// TIA Portal V20 export
// export: Created 2025-12-01T14:57:42.4272201Z, ExportSetting None, DisplayName Totally Integrated Automation Portal, DisplayVersion V20 Update 3, DisplayName TIA Portal Openness, DisplayVersion V20 Update 3, DisplayName TIA Portal Version Control Interface, DisplayVersion V20 Update 3, DisplayName STEP 7 Professional, DisplayVersion V20 Update 3, DisplayName STEP 7 Safety, DisplayVersion V20 Update 2, DisplayName WinCC Basic/Comfort/Advanced, DisplayVersion V20 Update 3, DisplayName WinCC Professional, DisplayVersion V20 Update 3, DisplayName WinCC Unified, DisplayVersion V20 Update 3
DATA_BLOCK "DB5_Emison"   // DB5
{ S7_Optimized_Access := 'FALSE' }
// stored: AutoNumber false
   VAR
      ByteLIbre_000 : Byte;
      RecepOK_M1 : Bool;
      PresNormal_M1 : Bool;
      Ausencia_M1 : Bool;
      PresBloqueo_M1 : Bool;
      Galibo_M1 : Bool;
      PresPreparada_M1 : Bool;
      PresMultiple_M1 : Bool;
      Bit_07_M1 : Bool;
      RecepOK_M2 : Bool;
      PresNormal_M2 : Bool;
      Ausencia_M2 : Bool;
      PresBloqueo_M2 : Bool;
      Galibo_M2 : Bool;
      PresPreparada_M2 : Bool;
      PresMultiple_M2 : Bool;
      Bit_07_M2 : Bool;
      RecepOK_M3 : Bool;
      PresNormal_M3 : Bool;
      Ausencia_M3 : Bool;
      PresBloqueo_M3 : Bool;
      Galibo_M3 : Bool;
      PresPreparada_M3 : Bool;
      PresMultiple_M3 : Bool;
      Bit_07_M3 : Bool;
      RecepOK_M4 : Bool;
      PresNormal_M4 : Bool;
      Ausencia_M4 : Bool;
      PresBloqueo_M4 : Bool;
      Galibo_M4 : Bool;
      PresPreparada_M4 : Bool;
      PresMultiple_M4 : Bool;
      Bit_07_M4 : Bool;
      RecepOK_M5 : Bool;
      PresNormal_M5 : Bool;
      Ausencia_M5 : Bool;
      PresBloqueo_M5 : Bool;
      Galibo_M5 : Bool;
      PresPreparada_M5 : Bool;
      PresMultiple_M5 : Bool;
      Bit_07_M5 : Bool;
      RecepOK_M6 : Bool;
      PresNormal_M6 : Bool;
      Ausencia_M6 : Bool;
      PresBloqueo_M6 : Bool;
      Galibo_M6 : Bool;
      PresPreparada_M6 : Bool;
      PresMultiple_M6 : Bool;
      Bit_07_M6 : Bool;
      RecepOK_M7 : Bool;
      PresNormal_M7 : Bool;
      Ausencia_M7 : Bool;
      PresBloqueo_M7 : Bool;
      Galibo_M7 : Bool;
      PresPreparada_M7 : Bool;
      PresMultiple_M7 : Bool;
      Bit_07_M7 : Bool;
      RecepOK_M8 : Bool;
      PresNormal_M8 : Bool;
      Ausencia_M8 : Bool;
      PresBloqueo_M8 : Bool;
      Galibo_M8 : Bool;
      PresPreparada_M8 : Bool;
      PresMultiple_M8 : Bool;
      Bit_07_M8 : Bool;
      RecepOK_M9 : Bool;
      PresNormal_M9 : Bool;
      Ausencia_M9 : Bool;
      PresBloqueo_M9 : Bool;
      Galibo_M9 : Bool;
      PresPreparada_M9 : Bool;
      PresMultiple_M9 : Bool;
      Bit_07_M9 : Bool;
      RecepOK_M10 : Bool;
      PresNormal_M10 : Bool;
      Ausencia_M10 : Bool;
      PresBloqueo_M10 : Bool;
      Galibo_M10 : Bool;
      PresPreparada_M10 : Bool;
      PresMultiple_M10 : Bool;
      Bit_07_M10 : Bool;
      RecepOK_M11 : Bool;
      PresNormal_M11 : Bool;
      Ausencia_M11 : Bool;
      PresBloqueo_M11 : Bool;
      Galibo_M11 : Bool;
      PresPreparada_M11 : Bool;
      PresMultiple_M11 : Bool;
      Bit_07_M11 : Bool;
      RecepOK_M12 : Bool;
      PresNormal_M12 : Bool;
      Ausencia_M12 : Bool;
      PresBloqueo_M12 : Bool;
      Galibo_M12 : Bool;
      PresPreparada_M12 : Bool;
      PresMultiple_M12 : Bool;
      Bit_07_M12 : Bool;
      RecepOK_M13 : Bool;
      PresNormal_M13 : Bool;
      Ausencia_M13 : Bool;
      PresBloqueo_M13 : Bool;
      Galibo_M13 : Bool;
      PresPreparada_M13 : Bool;
      PresMultiple_M13 : Bool;
      Bit_07_M13 : Bool;
      RecepOK_M14 : Bool;
      PresNormal_M14 : Bool;
      Ausencia_M14 : Bool;
      PresBloqueo_M14 : Bool;
      Galibo_M14 : Bool;
      PresPreparada_M14 : Bool;
      PresMultiple_M14 : Bool;
      Bit_07_M14 : Bool;
      RecepOK_M15 : Bool;
      PresNormal_M15 : Bool;
      Ausencia_M15 : Bool;
      PresBloqueo_M15 : Bool;
      Galibo_M15 : Bool;
      PresPreparada_M15 : Bool;
      PresMultiple_M15 : Bool;
      Bit_07_M15 : Bool;
      RecepOK_M16 : Bool;
      PresNormal_M16 : Bool;
      Ausencia_M16 : Bool;
      PresBloqueo_M16 : Bool;
      Galibo_M16 : Bool;
      PresPreparada_M16 : Bool;
      PresMultiple_M16 : Bool;
      Bit_07_M16 : Bool;
      RecepOK_M17 : Bool;
      PresNormal_M17 : Bool;
      Ausencia_M17 : Bool;
      PresBloqueo_M17 : Bool;
      Galibo_M17 : Bool;
      PresPreparada_M17 : Bool;
      PresMultiple_M17 : Bool;
      Bit_07_M17 : Bool;
      RecepOK_M18 : Bool;
      PresNormal_M18 : Bool;
      Ausencia_M18 : Bool;
      PresBloqueo_M18 : Bool;
      Galibo_M18 : Bool;
      PresPreparada_M18 : Bool;
      PresMultiple_M18 : Bool;
      Bit_07_M18 : Bool;
      RecepOK_M19 : Bool;
      PresNormal_M19 : Bool;
      Ausencia_M19 : Bool;
      PresBloqueo_M19 : Bool;
      Galibo_M19 : Bool;
      PresPreparada_M19 : Bool;
      PresMultiple_M19 : Bool;
      Bit_07_M19 : Bool;
      RecepOK_M20 : Bool;
      PresNormal_M20 : Bool;
      Ausencia_M20 : Bool;
      PresBloqueo_M20 : Bool;
      Galibo_M20 : Bool;
      PresPreparada_M20 : Bool;
      PresMultiple_M20 : Bool;
      Bit_07_M20 : Bool;
      RecepOK_M21 : Bool;
      PresNormal_M21 : Bool;
      Ausencia_M21 : Bool;
      PresBloqueo_M21 : Bool;
      Galibo_M21 : Bool;
      PresPreparada_M21 : Bool;
      PresMultiple_M21 : Bool;
      Bit_07_M21 : Bool;
      RecepOK_M22 : Bool;
      PresNormal_M22 : Bool;
      Ausencia_M22 : Bool;
      PresBloqueo_M22 : Bool;
      Galibo_M22 : Bool;
      PresPreparada_M22 : Bool;
      PresMultiple_M22 : Bool;
      Bit_07_M22 : Bool;
      RecepOK_M23 : Bool;
      PresNormal_M23 : Bool;
      Ausencia_M23 : Bool;
      PresBloqueo_M23 : Bool;
      Galibo_M23 : Bool;
      PresPreparada_M23 : Bool;
      PresMultiple_M23 : Bool;
      Bit_07_M23 : Bool;
      RecepOK_M24 : Bool;
      PresNormal_M24 : Bool;
      Ausencia_M24 : Bool;
      PresBloqueo_M24 : Bool;
      Galibo_M24 : Bool;
      PresPreparada_M24 : Bool;
      PresMultiple_M24 : Bool;
      Bit_07_M24 : Bool;
      RecepOK_M25 : Bool;
      PresNormal_M25 : Bool;
      Ausencia_M25 : Bool;
      PresBloqueo_M25 : Bool;
      Galibo_M25 : Bool;
      PresPreparada_M25 : Bool;
      PresMultiple_M25 : Bool;
      Bit_07_M25 : Bool;
      RecepOK_M26 : Bool;
      PresNormal_M26 : Bool;
      Ausencia_M26 : Bool;
      PresBloqueo_M26 : Bool;
      Galibo_M26 : Bool;
      PresPreparada_M26 : Bool;
      PresMultiple_M26 : Bool;
      Bit_07_M26 : Bool;
      RecepOK_M27 : Bool;
      PresNormal_M27 : Bool;
      Ausencia_M27 : Bool;
      PresBloqueo_M27 : Bool;
      Galibo_M27 : Bool;
      PresPreparada_M27 : Bool;
      PresMultiple_M27 : Bool;
      Bit_07_M27 : Bool;
      RecepOK_M28 : Bool;
      PresNormal_M28 : Bool;
      Ausencia_M28 : Bool;
      PresBloqueo_M28 : Bool;
      Galibo_M28 : Bool;
      PresPreparada_M28 : Bool;
      PresMultiple_M28 : Bool;
      Bit_07_M28 : Bool;
      RecepOK_M29 : Bool;
      PresNormal_M29 : Bool;
      Ausencia_M29 : Bool;
      PresBloqueo_M29 : Bool;
      Galibo_M29 : Bool;
      PresPreparada_M29 : Bool;
      PresMultiple_M29 : Bool;
      Bit_07_M29 : Bool;
      RecepOK_M30 : Bool;
      PresNormal_M30 : Bool;
      Ausencia_M30 : Bool;
      PresBloqueo_M30 : Bool;
      Galibo_M30 : Bool;
      PresPreparada_M30 : Bool;
      PresMultiple_M30 : Bool;
      Bit_07_M30 : Bool;
      RecepOK_M31 : Bool;
      PresNormal_M31 : Bool;
      Ausencia_M31 : Bool;
      PresBloqueo_M31 : Bool;
      Galibo_M31 : Bool;
      PresPreparada_M31 : Bool;
      PresMultiple_M31 : Bool;
      Bit_07_M31 : Bool;
      RecepOK_M32 : Bool;
      PresNormal_M32 : Bool;
      Ausencia_M32 : Bool;
      PresBloqueo_M32 : Bool;
      Galibo_M32 : Bool;
      PresPreparada_M32 : Bool;
      PresMultiple_M32 : Bool;
      Bit_07_M32 : Bool;
      RecepOK_M33 : Bool;
      PresNormal_M33 : Bool;
      Ausencia_M33 : Bool;
      PresBloqueo_M33 : Bool;
      Galibo_M33 : Bool;
      PresPreparada_M33 : Bool;
      PresMultiple_M33 : Bool;
      Bit_07_M33 : Bool;
      RecepOK_M34 : Bool;
      PresNormal_M34 : Bool;
      Ausencia_M34 : Bool;
      PresBloqueo_M34 : Bool;
      Galibo_M34 : Bool;
      PresPreparada_M34 : Bool;
      PresMultiple_M34 : Bool;
      Bit_07_M34 : Bool;
      RecepOK_M35 : Bool;
      PresNormal_M35 : Bool;
      Ausencia_M35 : Bool;
      PresBloqueo_M35 : Bool;
      Galibo_M35 : Bool;
      PresPreparada_M35 : Bool;
      PresMultiple_M35 : Bool;
      Bit_07_M35 : Bool;
      RecepOK_M36 : Bool;
      PresNormal_M36 : Bool;
      Ausencia_M36 : Bool;
      PresBloqueo_M36 : Bool;
      Galibo_M36 : Bool;
      PresPreparada_M36 : Bool;
      PresMultiple_M36 : Bool;
      Bit_07_M36 : Bool;
      RecepOK_M37 : Bool;
      PresNormal_M37 : Bool;
      Ausencia_M37 : Bool;
      PresBloqueo_M37 : Bool;
      Galibo_M37 : Bool;
      PresPreparada_M37 : Bool;
      PresMultiple_M37 : Bool;
      Bit_07_M37 : Bool;
      RecepOK_M38 : Bool;
      PresNormal_M38 : Bool;
      Ausencia_M38 : Bool;
      PresBloqueo_M38 : Bool;
      Galibo_M38 : Bool;
      PresPreparada_M38 : Bool;
      PresMultiple_M38 : Bool;
      Bit_07_M38 : Bool;
      RecepOK_M39 : Bool;
      PresNormal_M39 : Bool;
      Ausencia_M39 : Bool;
      PresBloqueo_M39 : Bool;
      Galibo_M39 : Bool;
      PresPreparada_M39 : Bool;
      PresMultiple_M39 : Bool;
      Bit_07_M39 : Bool;
      RecepOK_M40 : Bool;
      PresNormal_M40 : Bool;
      Ausencia_M40 : Bool;
      PresBloqueo_M40 : Bool;
      Galibo_M40 : Bool;
      PresPreparada_M40 : Bool;
      PresMultiple_M40 : Bool;
      Bit_07_M40 : Bool;
      RecepOK_M41 : Bool;
      PresNormal_M41 : Bool;
      Ausencia_M41 : Bool;
      PresBloqueo_M41 : Bool;
      Galibo_M41 : Bool;
      PresPreparada_M41 : Bool;
      PresMultiple_M41 : Bool;
      Bit_07_M41 : Bool;
      RecepOK_M42 : Bool;
      PresNormal_M42 : Bool;
      Ausencia_M42 : Bool;
      PresBloqueo_M42 : Bool;
      Galibo_M42 : Bool;
      PresPreparada_M42 : Bool;
      PresMultiple_M42 : Bool;
      Bit_07_M42 : Bool;
      RecepOK_M43 : Bool;
      PresNormal_M43 : Bool;
      Ausencia_M43 : Bool;
      PresBloqueo_M43 : Bool;
      Galibo_M43 : Bool;
      PresPreparada_M43 : Bool;
      PresMultiple_M43 : Bool;
      Bit_07_M43 : Bool;
      RecepOK_M44 : Bool;
      PresNormal_M44 : Bool;
      Ausencia_M44 : Bool;
      PresBloqueo_M44 : Bool;
      Galibo_M44 : Bool;
      PresPreparada_M44 : Bool;
      PresMultiple_M44 : Bool;
      Bit_07_M44 : Bool;
      RecepOK_M45 : Bool;
      PresNormal_M45 : Bool;
      Ausencia_M45 : Bool;
      PresBloqueo_M45 : Bool;
      Galibo_M45 : Bool;
      PresPreparada_M45 : Bool;
      PresMultiple_M45 : Bool;
      Bit_07_M45 : Bool;
      RecepOK_M46 : Bool;
      PresNormal_M46 : Bool;
      Ausencia_M46 : Bool;
      PresBloqueo_M46 : Bool;
      Galibo_M46 : Bool;
      PresPreparada_M46 : Bool;
      PresMultiple_M46 : Bool;
      Bit_07_M46 : Bool;
      RecepOK_M47 : Bool;
      PresNormal_M47 : Bool;
      Ausencia_M47 : Bool;
      PresBloqueo_M47 : Bool;
      Galibo_M47 : Bool;
      PresPreparada_M47 : Bool;
      PresMultiple_M47 : Bool;
      Bit_07_M47 : Bool;
      RecepOK_M48 : Bool;
      PresNormal_M48 : Bool;
      Ausencia_M48 : Bool;
      PresBloqueo_M48 : Bool;
      Galibo_M48 : Bool;
      PresPreparada_M48 : Bool;
      PresMultiple_M48 : Bool;
      Bit_07_M48 : Bool;
      RecepOK_M49 : Bool;
      PresNormal_M49 : Bool;
      Ausencia_M49 : Bool;
      PresBloqueo_M49 : Bool;
      Galibo_M49 : Bool;
      PresPreparada_M49 : Bool;
      PresMultiple_M49 : Bool;
      Bit_07_M49 : Bool;
      RecepOK_M50 : Bool;
      PresNormal_M50 : Bool;
      Ausencia_M50 : Bool;
      PresBloqueo_M50 : Bool;
      Galibo_M50 : Bool;
      PresPreparada_M50 : Bool;
      PresMultiple_M50 : Bool;
      Bit_07_M50 : Bool;
      RecepOK_M51 : Bool;
      PresNormal_M51 : Bool;
      Ausencia_M51 : Bool;
      PresBloqueo_M51 : Bool;
      Galibo_M51 : Bool;
      PresPreparada_M51 : Bool;
      PresMultiple_M51 : Bool;
      Bit_07_M51 : Bool;
      RecepOK_M52 : Bool;
      PresNormal_M52 : Bool;
      Ausencia_M52 : Bool;
      PresBloqueo_M52 : Bool;
      Galibo_M52 : Bool;
      PresPreparada_M52 : Bool;
      PresMultiple_M52 : Bool;
      Bit_07_M52 : Bool;
      RecepOK_M53 : Bool;
      PresNormal_M53 : Bool;
      Ausencia_M53 : Bool;
      PresBloqueo_M53 : Bool;
      Galibo_M53 : Bool;
      PresPreparada_M53 : Bool;
      PresMultiple_M53 : Bool;
      Bit_07_M53 : Bool;
      RecepOK_M54 : Bool;
      PresNormal_M54 : Bool;
      Ausencia_M54 : Bool;
      PresBloqueo_M54 : Bool;
      Galibo_M54 : Bool;
      PresPreparada_M54 : Bool;
      PresMultiple_M54 : Bool;
      Bit_07_M54 : Bool;
      RecepOK_M55 : Bool;
      PresNormal_M55 : Bool;
      Ausencia_M55 : Bool;
      PresBloqueo_M55 : Bool;
      Galibo_M55 : Bool;
      PresPreparada_M55 : Bool;
      PresMultiple_M55 : Bool;
      Bit_07_M55 : Bool;
      RecepOK_M56 : Bool;
      PresNormal_M56 : Bool;
      Ausencia_M56 : Bool;
      PresBloqueo_M56 : Bool;
      Galibo_M56 : Bool;
      PresPreparada_M56 : Bool;
      PresMultiple_M56 : Bool;
      Bit_07_M56 : Bool;
      RecepOK_M57 : Bool;
      PresNormal_M57 : Bool;
      Ausencia_M57 : Bool;
      PresBloqueo_M57 : Bool;
      Galibo_M57 : Bool;
      PresPreparada_M57 : Bool;
      PresMultiple_M57 : Bool;
      Bit_07_M57 : Bool;
      RecepOK_M58 : Bool;
      PresNormal_M58 : Bool;
      Ausencia_M58 : Bool;
      PresBloqueo_M58 : Bool;
      Galibo_M58 : Bool;
      PresPreparada_M58 : Bool;
      PresMultiple_M58 : Bool;
      Bit_07_M58 : Bool;
      RecepOK_M59 : Bool;
      PresNormal_M59 : Bool;
      Ausencia_M59 : Bool;
      PresBloqueo_M59 : Bool;
      Galibo_M59 : Bool;
      PresPreparada_M59 : Bool;
      PresMultiple_M59 : Bool;
      Bit_07_M59 : Bool;
      RecepOK_M60 : Bool;
      PresNormal_M60 : Bool;
      Ausencia_M60 : Bool;
      PresBloqueo_M60 : Bool;
      Galibo_M60 : Bool;
      PresPreparada_M60 : Bool;
      PresMultiple_M60 : Bool;
      Bit_07_M60 : Bool;
      RecepOK_M61 : Bool;
      PresNormal_M61 : Bool;
      Ausencia_M61 : Bool;
      PresBloqueo_M61 : Bool;
      Galibo_M61 : Bool;
      PresPreparada_M61 : Bool;
      PresMultiple_M61 : Bool;
      Bit_07_M61 : Bool;
      RecepOK_M62 : Bool;
      PresNormal_M62 : Bool;
      Ausencia_M62 : Bool;
      PresBloqueo_M62 : Bool;
      Galibo_M62 : Bool;
      PresPreparada_M62 : Bool;
      PresMultiple_M62 : Bool;
      Bit_07_M62 : Bool;
      RecepOK_M63 : Bool;
      PresNormal_M63 : Bool;
      Ausencia_M63 : Bool;
      PresBloqueo_M63 : Bool;
      Galibo_M63 : Bool;
      PresPreparada_M63 : Bool;
      PresMultiple_M63 : Bool;
      Bit_07_M63 : Bool;
      RecepOK_M64 : Bool;
      PresNormal_M64 : Bool;
      Ausencia_M64 : Bool;
      PresBloqueo_M64 : Bool;
      Galibo_M64 : Bool;
      PresPreparada_M64 : Bool;
      PresMultiple_M64 : Bool;
      Bit_07_M64 : Bool;
      RecepOK_M65 : Bool;
      PresNormal_M65 : Bool;
      Ausencia_M65 : Bool;
      PresBloqueo_M65 : Bool;
      Galibo_M65 : Bool;
      PresPreparada_M65 : Bool;
      PresMultiple_M65 : Bool;
      Bit_07_M65 : Bool;
      RecepOK_M66 : Bool;
      PresNormal_M66 : Bool;
      Ausencia_M66 : Bool;
      PresBloqueo_M66 : Bool;
      Galibo_M66 : Bool;
      PresPreparada_M66 : Bool;
      PresMultiple_M66 : Bool;
      Bit_07_M66 : Bool;
      RecepOK_M67 : Bool;
      PresNormal_M67 : Bool;
      Ausencia_M67 : Bool;
      PresBloqueo_M67 : Bool;
      Galibo_M67 : Bool;
      PresPreparada_M67 : Bool;
      PresMultiple_M67 : Bool;
      Bit_07_M67 : Bool;
      RecepOK_M68 : Bool;
      PresNormal_M68 : Bool;
      Ausencia_M68 : Bool;
      PresBloqueo_M68 : Bool;
      Galibo_M68 : Bool;
      PresPreparada_M68 : Bool;
      PresMultiple_M68 : Bool;
      Bit_07_M68 : Bool;
      RecepOK_M69 : Bool;
      PresNormal_M69 : Bool;
      Ausencia_M69 : Bool;
      PresBloqueo_M69 : Bool;
      Galibo_M69 : Bool;
      PresPreparada_M69 : Bool;
      PresMultiple_M69 : Bool;
      Bit_07_M69 : Bool;
      RecepOK_M70 : Bool;
      PresNormal_M70 : Bool;
      Ausencia_M70 : Bool;
      PresBloqueo_M70 : Bool;
      Galibo_M70 : Bool;
      PresPreparada_M70 : Bool;
      PresMultiple_M70 : Bool;
      Bit_07_M70 : Bool;
      RecepOK_M71 : Bool;
      PresNormal_M71 : Bool;
      Ausencia_M71 : Bool;
      PresBloqueo_M71 : Bool;
      Galibo_M71 : Bool;
      PresPreparada_M71 : Bool;
      PresMultiple_M71 : Bool;
      Bit_07_M71 : Bool;
      RecepOK_M72 : Bool;
      PresNormal_M72 : Bool;
      Ausencia_M72 : Bool;
      PresBloqueo_M72 : Bool;
      Galibo_M72 : Bool;
      PresPreparada_M72 : Bool;
      PresMultiple_M72 : Bool;
      Bit_07_M72 : Bool;
      RecepOK_M73 : Bool;
      PresNormal_M73 : Bool;
      Ausencia_M73 : Bool;
      PresBloqueo_M73 : Bool;
      Galibo_M73 : Bool;
      PresPreparada_M73 : Bool;
      PresMultiple_M73 : Bool;
      Bit_07_M73 : Bool;
      RecepOK_M74 : Bool;
      PresNormal_M74 : Bool;
      Ausencia_M74 : Bool;
      PresBloqueo_M74 : Bool;
      Galibo_M74 : Bool;
      PresPreparada_M74 : Bool;
      PresMultiple_M74 : Bool;
      Bit_07_M74 : Bool;
      RecepOK_M75 : Bool;
      PresNormal_M75 : Bool;
      Ausencia_M75 : Bool;
      PresBloqueo_M75 : Bool;
      Galibo_M75 : Bool;
      PresPreparada_M75 : Bool;
      PresMultiple_M75 : Bool;
      Bit_07_M75 : Bool;
      RecepOK_M76 : Bool;
      PresNormal_M76 : Bool;
      Ausencia_M76 : Bool;
      PresBloqueo_M76 : Bool;
      Galibo_M76 : Bool;
      PresPreparada_M76 : Bool;
      PresMultiple_M76 : Bool;
      Bit_07_M76 : Bool;
      RecepOK_M77 : Bool;
      PresNormal_M77 : Bool;
      Ausencia_M77 : Bool;
      PresBloqueo_M77 : Bool;
      Galibo_M77 : Bool;
      PresPreparada_M77 : Bool;
      PresMultiple_M77 : Bool;
      Bit_07_M77 : Bool;
      RecepOK_M78 : Bool;
      PresNormal_M78 : Bool;
      Ausencia_M78 : Bool;
      PresBloqueo_M78 : Bool;
      Galibo_M78 : Bool;
      PresPreparada_M78 : Bool;
      PresMultiple_M78 : Bool;
      Bit_07_M78 : Bool;
      RecepOK_M79 : Bool;
      PresNormal_M79 : Bool;
      Ausencia_M79 : Bool;
      PresBloqueo_M79 : Bool;
      Galibo_M79 : Bool;
      PresPreparada_M79 : Bool;
      PresMultiple_M79 : Bool;
      Bit_07_M79 : Bool;
      RecepOK_M80 : Bool;
      PresNormal_M80 : Bool;
      Ausencia_M80 : Bool;
      PresBloqueo_M80 : Bool;
      Galibo_M80 : Bool;
      PresPreparada_M80 : Bool;
      PresMultiple_M80 : Bool;
      Bit_07_M80 : Bool;
      RecepOK_M81 : Bool;
      PresNormal_M81 : Bool;
      Ausencia_M81 : Bool;
      PresBloqueo_M81 : Bool;
      Galibo_M81 : Bool;
      PresPreparada_M81 : Bool;
      PresMultiple_M81 : Bool;
      Bit_07_M81 : Bool;
      RecepOK_M82 : Bool;
      PresNormal_M82 : Bool;
      Ausencia_M82 : Bool;
      PresBloqueo_M82 : Bool;
      Galibo_M82 : Bool;
      PresPreparada_M82 : Bool;
      PresMultiple_M82 : Bool;
      Bit_07_M82 : Bool;
      RecepOK_M83 : Bool;
      PresNormal_M83 : Bool;
      Ausencia_M83 : Bool;
      PresBloqueo_M83 : Bool;
      Galibo_M83 : Bool;
      PresPreparada_M83 : Bool;
      PresMultiple_M83 : Bool;
      Bit_07_M83 : Bool;
      RecepOK_M84 : Bool;
      PresNormal_M84 : Bool;
      Ausencia_M84 : Bool;
      PresBloqueo_M84 : Bool;
      Galibo_M84 : Bool;
      PresPreparada_M84 : Bool;
      PresMultiple_M84 : Bool;
      Bit_07_M84 : Bool;
      RecepOK_M85 : Bool;
      PresNormal_M85 : Bool;
      Ausencia_M85 : Bool;
      PresBloqueo_M85 : Bool;
      Galibo_M85 : Bool;
      PresPreparada_M85 : Bool;
      PresMultiple_M85 : Bool;
      Bit_07_M85 : Bool;
      RecepOK_M86 : Bool;
      PresNormal_M86 : Bool;
      Ausencia_M86 : Bool;
      PresBloqueo_M86 : Bool;
      Galibo_M86 : Bool;
      PresPreparada_M86 : Bool;
      PresMultiple_M86 : Bool;
      Bit_07_M86 : Bool;
      RecepOK_M87 : Bool;
      PresNormal_M87 : Bool;
      Ausencia_M87 : Bool;
      PresBloqueo_M87 : Bool;
      Galibo_M87 : Bool;
      PresPreparada_M87 : Bool;
      PresMultiple_M87 : Bool;
      Bit_07_M87 : Bool;
      RecepOK_M88 : Bool;
      PresNormal_M88 : Bool;
      Ausencia_M88 : Bool;
      PresBloqueo_M88 : Bool;
      Galibo_M88 : Bool;
      PresPreparada_M88 : Bool;
      PresMultiple_M88 : Bool;
      Bit_07_M88 : Bool;
      RecepOK_M89 : Bool;
      PresNormal_M89 : Bool;
      Ausencia_M89 : Bool;
      PresBloqueo_M89 : Bool;
      Galibo_M89 : Bool;
      PresPreparada_M89 : Bool;
      PresMultiple_M89 : Bool;
      Bit_07_M89 : Bool;
      RecepOK_M90 : Bool;
      PresNormal_M90 : Bool;
      Ausencia_M90 : Bool;
      PresBloqueo_M90 : Bool;
      Galibo_M90 : Bool;
      PresPreparada_M90 : Bool;
      PresMultiple_M90 : Bool;
      Bit_07_M90 : Bool;
      RecepOK_M91 : Bool;
      PresNormal_M91 : Bool;
      Ausencia_M91 : Bool;
      PresBloqueo_M91 : Bool;
      Galibo_M91 : Bool;
      PresPreparada_M91 : Bool;
      PresMultiple_M91 : Bool;
      Bit_07_M91 : Bool;
      RecepOK_M92 : Bool;
      PresNormal_M92 : Bool;
      Ausencia_M92 : Bool;
      PresBloqueo_M92 : Bool;
      Galibo_M92 : Bool;
      PresPreparada_M92 : Bool;
      PresMultiple_M92 : Bool;
      Bit_07_M92 : Bool;
      RecepOK_M93 : Bool;
      PresNormal_M93 : Bool;
      Ausencia_M93 : Bool;
      PresBloqueo_M93 : Bool;
      Galibo_M93 : Bool;
      PresPreparada_M93 : Bool;
      PresMultiple_M93 : Bool;
      Bit_07_M93 : Bool;
      RecepOK_M94 : Bool;
      PresNormal_M94 : Bool;
      Ausencia_M94 : Bool;
      PresBloqueo_M94 : Bool;
      Galibo_M94 : Bool;
      PresPreparada_M94 : Bool;
      PresMultiple_M94 : Bool;
      Bit_07_M94 : Bool;
      RecepOK_M95 : Bool;
      PresNormal_M95 : Bool;
      Ausencia_M95 : Bool;
      PresBloqueo_M95 : Bool;
      Galibo_M95 : Bool;
      PresPreparada_M95 : Bool;
      PresMultiple_M95 : Bool;
      Bit_07_M95 : Bool;
      RecepOK_M96 : Bool;
      PresNormal_M96 : Bool;
      Ausencia_M96 : Bool;
      PresBloqueo_M96 : Bool;
      Galibo_M96 : Bool;
      PresPreparada_M96 : Bool;
      PresMultiple_M96 : Bool;
      Bit_07_M96 : Bool;
      RecepOK_M97 : Bool;
      PresNormal_M97 : Bool;
      Ausencia_M97 : Bool;
      PresBloqueo_M97 : Bool;
      Galibo_M97 : Bool;
      PresPreparada_M97 : Bool;
      PresMultiple_M97 : Bool;
      Bit_07_M97 : Bool;
      RecepOK_M98 : Bool;
      PresNormal_M98 : Bool;
      Ausencia_M98 : Bool;
      PresBloqueo_M98 : Bool;
      Galibo_M98 : Bool;
      PresPreparada_M98 : Bool;
      PresMultiple_M98 : Bool;
      Bit_07_M98 : Bool;
      RecepOK_M99 : Bool;
      PresNormal_M99 : Bool;
      Ausencia_M99 : Bool;
      PresBloqueo_M99 : Bool;
      Galibo_M99 : Bool;
      PresPreparada_M99 : Bool;
      PresMultiple_M99 : Bool;
      Bit_07_M99 : Bool;
      RecepOK_M100 : Bool;
      PresNormal_M100 : Bool;
      Ausencia_M100 : Bool;
      PresBloqueo_M100 : Bool;
      Galibo_M100 : Bool;
      PresPreparada_M100 : Bool;
      PresMultiple_M100 : Bool;
      Bit_07_M100 : Bool;
      RecepOK_M101 : Bool;
      PresNormal_M101 : Bool;
      Ausencia_M101 : Bool;
      PresBloqueo_M101 : Bool;
      Galibo_M101 : Bool;
      PresPreparada_M101 : Bool;
      PresMultiple_M101 : Bool;
      Bit_07_M101 : Bool;
      RecepOK_M102 : Bool;
      PresNormal_M102 : Bool;
      Ausencia_M102 : Bool;
      PresBloqueo_M102 : Bool;
      Galibo_M102 : Bool;
      PresPreparada_M102 : Bool;
      PresMultiple_M102 : Bool;
      Bit_07_M102 : Bool;
      RecepOK_M103 : Bool;
      PresNormal_M103 : Bool;
      Ausencia_M103 : Bool;
      PresBloqueo_M103 : Bool;
      Galibo_M103 : Bool;
      PresPreparada_M103 : Bool;
      PresMultiple_M103 : Bool;
      Bit_07_M103 : Bool;
      RecepOK_M104 : Bool;
      PresNormal_M104 : Bool;
      Ausencia_M104 : Bool;
      PresBloqueo_M104 : Bool;
      Galibo_M104 : Bool;
      PresPreparada_M104 : Bool;
      PresMultiple_M104 : Bool;
      Bit_07_M104 : Bool;
      RecepOK_M105 : Bool;
      PresNormal_M105 : Bool;
      Ausencia_M105 : Bool;
      PresBloqueo_M105 : Bool;
      Galibo_M105 : Bool;
      PresPreparada_M105 : Bool;
      PresMultiple_M105 : Bool;
      Bit_07_M105 : Bool;
      RecepOK_M106 : Bool;
      PresNormal_M106 : Bool;
      Ausencia_M106 : Bool;
      PresBloqueo_M106 : Bool;
      Galibo_M106 : Bool;
      PresPreparada_M106 : Bool;
      PresMultiple_M106 : Bool;
      Bit_07_M106 : Bool;
      RecepOK_M107 : Bool;
      PresNormal_M107 : Bool;
      Ausencia_M107 : Bool;
      PresBloqueo_M107 : Bool;
      Galibo_M107 : Bool;
      PresPreparada_M107 : Bool;
      PresMultiple_M107 : Bool;
      Bit_07_M107 : Bool;
      RecepOK_M108 : Bool;
      PresNormal_M108 : Bool;
      Ausencia_M108 : Bool;
      PresBloqueo_M108 : Bool;
      Galibo_M108 : Bool;
      PresPreparada_M108 : Bool;
      PresMultiple_M108 : Bool;
      Bit_07_M108 : Bool;
      RecepOK_M109 : Bool;
      PresNormal_M109 : Bool;
      Ausencia_M109 : Bool;
      PresBloqueo_M109 : Bool;
      Galibo_M109 : Bool;
      PresPreparada_M109 : Bool;
      PresMultiple_M109 : Bool;
      Bit_07_M109 : Bool;
      RecepOK_M110 : Bool;
      PresNormal_M110 : Bool;
      Ausencia_M110 : Bool;
      PresBloqueo_M110 : Bool;
      Galibo_M110 : Bool;
      PresPreparada_M110 : Bool;
      PresMultiple_M110 : Bool;
      Bit_07_M110 : Bool;
      RecepOK_M111 : Bool;
      PresNormal_M111 : Bool;
      Ausencia_M111 : Bool;
      PresBloqueo_M111 : Bool;
      Galibo_M111 : Bool;
      PresPreparada_M111 : Bool;
      PresMultiple_M111 : Bool;
      Bit_07_M111 : Bool;
      RecepOK_M112 : Bool;
      PresNormal_M112 : Bool;
      Ausencia_M112 : Bool;
      PresBloqueo_M112 : Bool;
      Galibo_M112 : Bool;
      PresPreparada_M112 : Bool;
      PresMultiple_M112 : Bool;
      Bit_07_M112 : Bool;
      RecepOK_M113 : Bool;
      PresNormal_M113 : Bool;
      Ausencia_M113 : Bool;
      PresBloqueo_M113 : Bool;
      Galibo_M113 : Bool;
      PresPreparada_M113 : Bool;
      PresMultiple_M113 : Bool;
      Bit_07_M113 : Bool;
      RecepOK_M114 : Bool;
      PresNormal_M114 : Bool;
      Ausencia_M114 : Bool;
      PresBloqueo_M114 : Bool;
      Galibo_M114 : Bool;
      PresPreparada_M114 : Bool;
      PresMultiple_M114 : Bool;
      Bit_07_M114 : Bool;
      RecepOK_M115 : Bool;
      PresNormal_M115 : Bool;
      Ausencia_M115 : Bool;
      PresBloqueo_M115 : Bool;
      Galibo_M115 : Bool;
      PresPreparada_M115 : Bool;
      PresMultiple_M115 : Bool;
      Bit_07_M115 : Bool;
      RecepOK_M116 : Bool;
      PresNormal_M116 : Bool;
      Ausencia_M116 : Bool;
      PresBloqueo_M116 : Bool;
      Galibo_M116 : Bool;
      PresPreparada_M116 : Bool;
      PresMultiple_M116 : Bool;
      Bit_07_M116 : Bool;
      RecepOK_M117 : Bool;
      PresNormal_M117 : Bool;
      Ausencia_M117 : Bool;
      PresBloqueo_M117 : Bool;
      Galibo_M117 : Bool;
      PresPreparada_M117 : Bool;
      PresMultiple_M117 : Bool;
      Bit_07_M117 : Bool;
      RecepOK_M118 : Bool;
      PresNormal_M118 : Bool;
      Ausencia_M118 : Bool;
      PresBloqueo_M118 : Bool;
      Galibo_M118 : Bool;
      PresPreparada_M118 : Bool;
      PresMultiple_M118 : Bool;
      Bit_07_M118 : Bool;
      RecepOK_M119 : Bool;
      PresNormal_M119 : Bool;
      Ausencia_M119 : Bool;
      PresBloqueo_M119 : Bool;
      Galibo_M119 : Bool;
      PresPreparada_M119 : Bool;
      PresMultiple_M119 : Bool;
      Bit_07_M119 : Bool;
      RecepOK_M120 : Bool;
      PresNormal_M120 : Bool;
      Ausencia_M120 : Bool;
      PresBloqueo_M120 : Bool;
      Galibo_M120 : Bool;
      PresPreparada_M120 : Bool;
      PresMultiple_M120 : Bool;
      Bit_07_M120 : Bool;
      RecepOK_M121 : Bool;
      PresNormal_M121 : Bool;
      Ausencia_M121 : Bool;
      PresBloqueo_M121 : Bool;
      Galibo_M121 : Bool;
      PresPreparada_M121 : Bool;
      PresMultiple_M121 : Bool;
      Bit_07_M121 : Bool;
      RecepOK_M122 : Bool;
      PresNormal_M122 : Bool;
      Ausencia_M122 : Bool;
      PresBloqueo_M122 : Bool;
      Galibo_M122 : Bool;
      PresPreparada_M122 : Bool;
      PresMultiple_M122 : Bool;
      Bit_07_M122 : Bool;
      RecepOK_M123 : Bool;
      PresNormal_M123 : Bool;
      Ausencia_M123 : Bool;
      PresBloqueo_M123 : Bool;
      Galibo_M123 : Bool;
      PresPreparada_M123 : Bool;
      PresMultiple_M123 : Bool;
      Bit_07_M123 : Bool;
      RecepOK_M124 : Bool;
      PresNormal_M124 : Bool;
      Ausencia_M124 : Bool;
      PresBloqueo_M124 : Bool;
      Galibo_M124 : Bool;
      PresPreparada_M124 : Bool;
      PresMultiple_M124 : Bool;
      Bit_07_M124 : Bool;
      RecepOK_M125 : Bool;
      PresNormal_M125 : Bool;
      Ausencia_M125 : Bool;
      PresBloqueo_M125 : Bool;
      Galibo_M125 : Bool;
      PresPreparada_M125 : Bool;
      PresMultiple_M125 : Bool;
      Bit_07_M125 : Bool;
      RecepOK_M126 : Bool;
      PresNormal_M126 : Bool;
      Ausencia_M126 : Bool;
      PresBloqueo_M126 : Bool;
      Galibo_M126 : Bool;
      PresPreparada_M126 : Bool;
      PresMultiple_M126 : Bool;
      Bit_07_M126 : Bool;
      RecepOK_M127 : Bool;
      PresNormal_M127 : Bool;
      Ausencia_M127 : Bool;
      PresBloqueo_M127 : Bool;
      Galibo_M127 : Bool;
      PresPreparada_M127 : Bool;
      PresMultiple_M127 : Bool;
      Bit_07_M127 : Bool;
      RecepOK_M128 : Bool;
      PresNormal_M128 : Bool;
      Ausencia_M128 : Bool;
      PresBloqueo_M128 : Bool;
      Galibo_M128 : Bool;
      PresPreparada_M128 : Bool;
      PresMultiple_M128 : Bool;
      Bit_07_M128 : Bool;
      RecepOK_M129 : Bool;
      PresNormal_M129 : Bool;
      Ausencia_M129 : Bool;
      PresBloqueo_M129 : Bool;
      Galibo_M129 : Bool;
      PresPreparada_M129 : Bool;
      PresMultiple_M129 : Bool;
      Bit_07_M129 : Bool;
      RecepOK_M130 : Bool;
      PresNormal_M130 : Bool;
      Ausencia_M130 : Bool;
      PresBloqueo_M130 : Bool;
      Galibo_M130 : Bool;
      PresPreparada_M130 : Bool;
      PresMultiple_M130 : Bool;
      Bit_07_M130 : Bool;
      RecepOK_M131 : Bool;
      PresNormal_M131 : Bool;
      Ausencia_M131 : Bool;
      PresBloqueo_M131 : Bool;
      Galibo_M131 : Bool;
      PresPreparada_M131 : Bool;
      PresMultiple_M131 : Bool;
      Bit_07_M131 : Bool;
      RecepOK_M132 : Bool;
      PresNormal_M132 : Bool;
      Ausencia_M132 : Bool;
      PresBloqueo_M132 : Bool;
      Galibo_M132 : Bool;
      PresPreparada_M132 : Bool;
      PresMultiple_M132 : Bool;
      Bit_07_M132 : Bool;
      RecepOK_M133 : Bool;
      PresNormal_M133 : Bool;
      Ausencia_M133 : Bool;
      PresBloqueo_M133 : Bool;
      Galibo_M133 : Bool;
      PresPreparada_M133 : Bool;
      PresMultiple_M133 : Bool;
      Bit_07_M133 : Bool;
      RecepOK_M134 : Bool;
      PresNormal_M134 : Bool;
      Ausencia_M134 : Bool;
      PresBloqueo_M134 : Bool;
      Galibo_M134 : Bool;
      PresPreparada_M134 : Bool;
      PresMultiple_M134 : Bool;
      Bit_07_M134 : Bool;
      RecepOK_M135 : Bool;
      PresNormal_M135 : Bool;
      Ausencia_M135 : Bool;
      PresBloqueo_M135 : Bool;
      Galibo_M135 : Bool;
      PresPreparada_M135 : Bool;
      PresMultiple_M135 : Bool;
      Bit_07_M135 : Bool;
      RecepOK_M136 : Bool;
      PresNormal_M136 : Bool;
      Ausencia_M136 : Bool;
      PresBloqueo_M136 : Bool;
      Galibo_M136 : Bool;
      PresPreparada_M136 : Bool;
      PresMultiple_M136 : Bool;
      Bit_07_M136 : Bool;
      RecepOK_M137 : Bool;
      PresNormal_M137 : Bool;
      Ausencia_M137 : Bool;
      PresBloqueo_M137 : Bool;
      Galibo_M137 : Bool;
      PresPreparada_M137 : Bool;
      PresMultiple_M137 : Bool;
      Bit_07_M137 : Bool;
      RecepOK_M138 : Bool;
      PresNormal_M138 : Bool;
      Ausencia_M138 : Bool;
      PresBloqueo_M138 : Bool;
      Galibo_M138 : Bool;
      PresPreparada_M138 : Bool;
      PresMultiple_M138 : Bool;
      Bit_07_M138 : Bool;
      RecepOK_M139 : Bool;
      PresNormal_M139 : Bool;
      Ausencia_M139 : Bool;
      PresBloqueo_M139 : Bool;
      Galibo_M139 : Bool;
      PresPreparada_M139 : Bool;
      PresMultiple_M139 : Bool;
      Bit_07_M139 : Bool;
      RecepOK_M140 : Bool;
      PresNormal_M140 : Bool;
      Ausencia_M140 : Bool;
      PresBloqueo_M140 : Bool;
      Galibo_M140 : Bool;
      PresPreparada_M140 : Bool;
      PresMultiple_M140 : Bool;
      Bit_07_M140 : Bool;
      RecepOK_M141 : Bool;
      PresNormal_M141 : Bool;
      Ausencia_M141 : Bool;
      PresBloqueo_M141 : Bool;
      Galibo_M141 : Bool;
      PresPreparada_M141 : Bool;
      PresMultiple_M141 : Bool;
      Bit_07_M141 : Bool;
      RecepOK_M142 : Bool;
      PresNormal_M142 : Bool;
      Ausencia_M142 : Bool;
      PresBloqueo_M142 : Bool;
      Galibo_M142 : Bool;
      PresPreparada_M142 : Bool;
      PresMultiple_M142 : Bool;
      Bit_07_M142 : Bool;
      RecepOK_M143 : Bool;
      PresNormal_M143 : Bool;
      Ausencia_M143 : Bool;
      PresBloqueo_M143 : Bool;
      Galibo_M143 : Bool;
      PresPreparada_M143 : Bool;
      PresMultiple_M143 : Bool;
      Bit_07_M143 : Bool;
      RecepOK_M144 : Bool;
      PresNormal_M144 : Bool;
      Ausencia_M144 : Bool;
      PresBloqueo_M144 : Bool;
      Galibo_M144 : Bool;
      PresPreparada_M144 : Bool;
      PresMultiple_M144 : Bool;
      Bit_07_M144 : Bool;
      RecepOK_M145 : Bool;
      PresNormal_M145 : Bool;
      Ausencia_M145 : Bool;
      PresBloqueo_M145 : Bool;
      Galibo_M145 : Bool;
      PresPreparada_M145 : Bool;
      PresMultiple_M145 : Bool;
      Bit_07_M145 : Bool;
      RecepOK_M146 : Bool;
      PresNormal_M146 : Bool;
      Ausencia_M146 : Bool;
      PresBloqueo_M146 : Bool;
      Galibo_M146 : Bool;
      PresPreparada_M146 : Bool;
      PresMultiple_M146 : Bool;
      Bit_07_M146 : Bool;
      RecepOK_M147 : Bool;
      PresNormal_M147 : Bool;
      Ausencia_M147 : Bool;
      PresBloqueo_M147 : Bool;
      Galibo_M147 : Bool;
      PresPreparada_M147 : Bool;
      PresMultiple_M147 : Bool;
      Bit_07_M147 : Bool;
      RecepOK_M148 : Bool;
      PresNormal_M148 : Bool;
      Ausencia_M148 : Bool;
      PresBloqueo_M148 : Bool;
      Galibo_M148 : Bool;
      PresPreparada_M148 : Bool;
      PresMultiple_M148 : Bool;
      Bit_07_M148 : Bool;
      RecepOK_M149 : Bool;
      PresNormal_M149 : Bool;
      Ausencia_M149 : Bool;
      PresBloqueo_M149 : Bool;
      Galibo_M149 : Bool;
      PresPreparada_M149 : Bool;
      PresMultiple_M149 : Bool;
      Bit_07_M149 : Bool;
      RecepOK_M150 : Bool;
      PresNormal_M150 : Bool;
      Ausencia_M150 : Bool;
      PresBloqueo_M150 : Bool;
      Galibo_M150 : Bool;
      PresPreparada_M150 : Bool;
      PresMultiple_M150 : Bool;
      Bit_07_M150 : Bool;
      RecepOK_M151 : Bool;
      PresNormal_M151 : Bool;
      Ausencia_M151 : Bool;
      PresBloqueo_M151 : Bool;
      Galibo_M151 : Bool;
      PresPreparada_M151 : Bool;
      PresMultiple_M151 : Bool;
      Bit_07_M151 : Bool;
      RecepOK_M152 : Bool;
      PresNormal_M152 : Bool;
      Ausencia_M152 : Bool;
      PresBloqueo_M152 : Bool;
      Galibo_M152 : Bool;
      PresPreparada_M152 : Bool;
      PresMultiple_M152 : Bool;
      Bit_07_M152 : Bool;
      RecepOK_M153 : Bool;
      PresNormal_M153 : Bool;
      Ausencia_M153 : Bool;
      PresBloqueo_M153 : Bool;
      Galibo_M153 : Bool;
      PresPreparada_M153 : Bool;
      PresMultiple_M153 : Bool;
      Bit_07_M153 : Bool;
      RecepOK_M154 : Bool;
      PresNormal_M154 : Bool;
      Ausencia_M154 : Bool;
      PresBloqueo_M154 : Bool;
      Galibo_M154 : Bool;
      PresPreparada_M154 : Bool;
      PresMultiple_M154 : Bool;
      Bit_07_M154 : Bool;
      RecepOK_M155 : Bool;
      PresNormal_M155 : Bool;
      Ausencia_M155 : Bool;
      PresBloqueo_M155 : Bool;
      Galibo_M155 : Bool;
      PresPreparada_M155 : Bool;
      PresMultiple_M155 : Bool;
      Bit_07_M155 : Bool;
      RecepOK_M156 : Bool;
      PresNormal_M156 : Bool;
      Ausencia_M156 : Bool;
      PresBloqueo_M156 : Bool;
      Galibo_M156 : Bool;
      PresPreparada_M156 : Bool;
      PresMultiple_M156 : Bool;
      Bit_07_M156 : Bool;
      RecepOK_M157 : Bool;
      PresNormal_M157 : Bool;
      Ausencia_M157 : Bool;
      PresBloqueo_M157 : Bool;
      Galibo_M157 : Bool;
      PresPreparada_M157 : Bool;
      PresMultiple_M157 : Bool;
      Bit_07_M157 : Bool;
      RecepOK_M158 : Bool;
      PresNormal_M158 : Bool;
      Ausencia_M158 : Bool;
      PresBloqueo_M158 : Bool;
      Galibo_M158 : Bool;
      PresPreparada_M158 : Bool;
      PresMultiple_M158 : Bool;
      Bit_07_M158 : Bool;
      RecepOK_M159 : Bool;
      PresNormal_M159 : Bool;
      Ausencia_M159 : Bool;
      PresBloqueo_M159 : Bool;
      Galibo_M159 : Bool;
      PresPreparada_M159 : Bool;
      PresMultiple_M159 : Bool;
      Bit_07_M159 : Bool;
      RecepOK_M160 : Bool;
      PresNormal_M160 : Bool;
      Ausencia_M160 : Bool;
      PresBloqueo_M160 : Bool;
      Galibo_M160 : Bool;
      PresPreparada_M160 : Bool;
      PresMultiple_M160 : Bool;
      Bit_07_M160 : Bool;
      RecepOK_M161 : Bool;
      PresNormal_M161 : Bool;
      Ausencia_M161 : Bool;
      PresBloqueo_M161 : Bool;
      Galibo_M161 : Bool;
      PresPreparada_M161 : Bool;
      PresMultiple_M161 : Bool;
      Bit_07_M161 : Bool;
      RecepOK_M162 : Bool;
      PresNormal_M162 : Bool;
      Ausencia_M162 : Bool;
      PresBloqueo_M162 : Bool;
      Galibo_M162 : Bool;
      PresPreparada_M162 : Bool;
      PresMultiple_M162 : Bool;
      Bit_07_M162 : Bool;
      RecepOK_M163 : Bool;
      PresNormal_M163 : Bool;
      Ausencia_M163 : Bool;
      PresBloqueo_M163 : Bool;
      Galibo_M163 : Bool;
      PresPreparada_M163 : Bool;
      PresMultiple_M163 : Bool;
      Bit_07_M163 : Bool;
      RecepOK_M164 : Bool;
      PresNormal_M164 : Bool;
      Ausencia_M164 : Bool;
      PresBloqueo_M164 : Bool;
      Galibo_M164 : Bool;
      PresPreparada_M164 : Bool;
      PresMultiple_M164 : Bool;
      Bit_07_M164 : Bool;
      RecepOK_M165 : Bool;
      PresNormal_M165 : Bool;
      Ausencia_M165 : Bool;
      PresBloqueo_M165 : Bool;
      Galibo_M165 : Bool;
      PresPreparada_M165 : Bool;
      PresMultiple_M165 : Bool;
      Bit_07_M165 : Bool;
      RecepOK_M166 : Bool;
      PresNormal_M166 : Bool;
      Ausencia_M166 : Bool;
      PresBloqueo_M166 : Bool;
      Galibo_M166 : Bool;
      PresPreparada_M166 : Bool;
      PresMultiple_M166 : Bool;
      Bit_07_M166 : Bool;
      RecepOK_M167 : Bool;
      PresNormal_M167 : Bool;
      Ausencia_M167 : Bool;
      PresBloqueo_M167 : Bool;
      Galibo_M167 : Bool;
      PresPreparada_M167 : Bool;
      PresMultiple_M167 : Bool;
      Bit_07_M167 : Bool;
      RecepOK_M168 : Bool;
      PresNormal_M168 : Bool;
      Ausencia_M168 : Bool;
      PresBloqueo_M168 : Bool;
      Galibo_M168 : Bool;
      PresPreparada_M168 : Bool;
      PresMultiple_M168 : Bool;
      Bit_07_M168 : Bool;
      RecepOK_M169 : Bool;
      PresNormal_M169 : Bool;
      Ausencia_M169 : Bool;
      PresBloqueo_M169 : Bool;
      Galibo_M169 : Bool;
      PresPreparada_M169 : Bool;
      PresMultiple_M169 : Bool;
      Bit_07_M169 : Bool;
      RecepOK_M170 : Bool;
      PresNormal_M170 : Bool;
      Ausencia_M170 : Bool;
      PresBloqueo_M170 : Bool;
      Galibo_M170 : Bool;
      PresPreparada_M170 : Bool;
      PresMultiple_M170 : Bool;
      Bit_07_M170 : Bool;
      RecepOK_M171 : Bool;
      PresNormal_M171 : Bool;
      Ausencia_M171 : Bool;
      PresBloqueo_M171 : Bool;
      Galibo_M171 : Bool;
      PresPreparada_M171 : Bool;
      PresMultiple_M171 : Bool;
      Bit_07_M171 : Bool;
      RecepOK_M172 : Bool;
      PresNormal_M172 : Bool;
      Ausencia_M172 : Bool;
      PresBloqueo_M172 : Bool;
      Galibo_M172 : Bool;
      PresPreparada_M172 : Bool;
      PresMultiple_M172 : Bool;
      Bit_07_M172 : Bool;
      RecepOK_M173 : Bool;
      PresNormal_M173 : Bool;
      Ausencia_M173 : Bool;
      PresBloqueo_M173 : Bool;
      Galibo_M173 : Bool;
      PresPreparada_M173 : Bool;
      PresMultiple_M173 : Bool;
      Bit_07_M173 : Bool;
      RecepOK_M174 : Bool;
      PresNormal_M174 : Bool;
      Ausencia_M174 : Bool;
      PresBloqueo_M174 : Bool;
      Galibo_M174 : Bool;
      PresPreparada_M174 : Bool;
      PresMultiple_M174 : Bool;
      Bit_07_M174 : Bool;
      RecepOK_M175 : Bool;
      PresNormal_M175 : Bool;
      Ausencia_M175 : Bool;
      PresBloqueo_M175 : Bool;
      Galibo_M175 : Bool;
      PresPreparada_M175 : Bool;
      PresMultiple_M175 : Bool;
      Bit_07_M175 : Bool;
      RecepOK_M176 : Bool;
      PresNormal_M176 : Bool;
      Ausencia_M176 : Bool;
      PresBloqueo_M176 : Bool;
      Galibo_M176 : Bool;
      PresPreparada_M176 : Bool;
      PresMultiple_M176 : Bool;
      Bit_07_M176 : Bool;
      RecepOK_M177 : Bool;
      PresNormal_M177 : Bool;
      Ausencia_M177 : Bool;
      PresBloqueo_M177 : Bool;
      Galibo_M177 : Bool;
      PresPreparada_M177 : Bool;
      PresMultiple_M177 : Bool;
      Bit_07_M177 : Bool;
      RecepOK_M178 : Bool;
      PresNormal_M178 : Bool;
      Ausencia_M178 : Bool;
      PresBloqueo_M178 : Bool;
      Galibo_M178 : Bool;
      PresPreparada_M178 : Bool;
      PresMultiple_M178 : Bool;
      Bit_07_M178 : Bool;
      RecepOK_M179 : Bool;
      PresNormal_M179 : Bool;
      Ausencia_M179 : Bool;
      PresBloqueo_M179 : Bool;
      Galibo_M179 : Bool;
      PresPreparada_M179 : Bool;
      PresMultiple_M179 : Bool;
      Bit_07_M179 : Bool;
      RecepOK_M180 : Bool;
      PresNormal_M180 : Bool;
      Ausencia_M180 : Bool;
      PresBloqueo_M180 : Bool;
      Galibo_M180 : Bool;
      PresPreparada_M180 : Bool;
      PresMultiple_M180 : Bool;
      Bit_07_M180 : Bool;
      RecepOK_M181 : Bool;
      PresNormal_M181 : Bool;
      Ausencia_M181 : Bool;
      PresBloqueo_M181 : Bool;
      Galibo_M181 : Bool;
      PresPreparada_M181 : Bool;
      PresMultiple_M181 : Bool;
      Bit_07_M181 : Bool;
      RecepOK_M182 : Bool;
      PresNormal_M182 : Bool;
      Ausencia_M182 : Bool;
      PresBloqueo_M182 : Bool;
      Galibo_M182 : Bool;
      PresPreparada_M182 : Bool;
      PresMultiple_M182 : Bool;
      Bit_07_M182 : Bool;
      RecepOK_M183 : Bool;
      PresNormal_M183 : Bool;
      Ausencia_M183 : Bool;
      PresBloqueo_M183 : Bool;
      Galibo_M183 : Bool;
      PresPreparada_M183 : Bool;
      PresMultiple_M183 : Bool;
      Bit_07_M183 : Bool;
      RecepOK_M184 : Bool;
      PresNormal_M184 : Bool;
      Ausencia_M184 : Bool;
      PresBloqueo_M184 : Bool;
      Galibo_M184 : Bool;
      PresPreparada_M184 : Bool;
      PresMultiple_M184 : Bool;
      Bit_07_M184 : Bool;
      RecepOK_M185 : Bool;
      PresNormal_M185 : Bool;
      Ausencia_M185 : Bool;
      PresBloqueo_M185 : Bool;
      Galibo_M185 : Bool;
      PresPreparada_M185 : Bool;
      PresMultiple_M185 : Bool;
      Bit_07_M185 : Bool;
      RecepOK_M186 : Bool;
      PresNormal_M186 : Bool;
      Ausencia_M186 : Bool;
      PresBloqueo_M186 : Bool;
      Galibo_M186 : Bool;
      PresPreparada_M186 : Bool;
      PresMultiple_M186 : Bool;
      Bit_07_M186 : Bool;
      RecepOK_M187 : Bool;
      PresNormal_M187 : Bool;
      Ausencia_M187 : Bool;
      PresBloqueo_M187 : Bool;
      Galibo_M187 : Bool;
      PresPreparada_M187 : Bool;
      PresMultiple_M187 : Bool;
      Bit_07_M187 : Bool;
      RecepOK_M188 : Bool;
      PresNormal_M188 : Bool;
      Ausencia_M188 : Bool;
      PresBloqueo_M188 : Bool;
      Galibo_M188 : Bool;
      PresPreparada_M188 : Bool;
      PresMultiple_M188 : Bool;
      Bit_07_M188 : Bool;
      RecepOK_M189 : Bool;
      PresNormal_M189 : Bool;
      Ausencia_M189 : Bool;
      PresBloqueo_M189 : Bool;
      Galibo_M189 : Bool;
      PresPreparada_M189 : Bool;
      PresMultiple_M189 : Bool;
      Bit_07_M189 : Bool;
      RecepOK_M190 : Bool;
      PresNormal_M190 : Bool;
      Ausencia_M190 : Bool;
      PresBloqueo_M190 : Bool;
      Galibo_M190 : Bool;
      PresPreparada_M190 : Bool;
      PresMultiple_M190 : Bool;
      Bit_07_M190 : Bool;
      RecepOK_M191 : Bool;
      PresNormal_M191 : Bool;
      Ausencia_M191 : Bool;
      PresBloqueo_M191 : Bool;
      Galibo_M191 : Bool;
      PresPreparada_M191 : Bool;
      PresMultiple_M191 : Bool;
      Bit_07_M191 : Bool;
      RecepOK_M192 : Bool;
      PresNormal_M192 : Bool;
      Ausencia_M192 : Bool;
      PresBloqueo_M192 : Bool;
      Galibo_M192 : Bool;
      PresPreparada_M192 : Bool;
      PresMultiple_M192 : Bool;
      Bit_07_M192 : Bool;
      RecepOK_M193 : Bool;
      PresNormal_M193 : Bool;
      Ausencia_M193 : Bool;
      PresBloqueo_M193 : Bool;
      Galibo_M193 : Bool;
      PresPreparada_M193 : Bool;
      PresMultiple_M193 : Bool;
      Bit_07_M193 : Bool;
      RecepOK_M194 : Bool;
      PresNormal_M194 : Bool;
      Ausencia_M194 : Bool;
      PresBloqueo_M194 : Bool;
      Galibo_M194 : Bool;
      PresPreparada_M194 : Bool;
      PresMultiple_M194 : Bool;
      Bit_07_M194 : Bool;
      RecepOK_M195 : Bool;
      PresNormal_M195 : Bool;
      Ausencia_M195 : Bool;
      PresBloqueo_M195 : Bool;
      Galibo_M195 : Bool;
      PresPreparada_M195 : Bool;
      PresMultiple_M195 : Bool;
      Bit_07_M195 : Bool;
      RecepOK_M196 : Bool;
      PresNormal_M196 : Bool;
      Ausencia_M196 : Bool;
      PresBloqueo_M196 : Bool;
      Galibo_M196 : Bool;
      PresPreparada_M196 : Bool;
      PresMultiple_M196 : Bool;
      Bit_07_M196 : Bool;
      RecepOK_M197 : Bool;
      PresNormal_M197 : Bool;
      Ausencia_M197 : Bool;
      PresBloqueo_M197 : Bool;
      Galibo_M197 : Bool;
      PresPreparada_M197 : Bool;
      PresMultiple_M197 : Bool;
      Bit_07_M197 : Bool;
      RecepOK_M198 : Bool;
      PresNormal_M198 : Bool;
      Ausencia_M198 : Bool;
      PresBloqueo_M198 : Bool;
      Galibo_M198 : Bool;
      PresPreparada_M198 : Bool;
      PresMultiple_M198 : Bool;
      Bit_07_M198 : Bool;
      RecepOK_M199 : Bool;
      PresNormal_M199 : Bool;
      Ausencia_M199 : Bool;
      PresBloqueo_M199 : Bool;
      Galibo_M199 : Bool;
      PresPreparada_M199 : Bool;
      PresMultiple_M199 : Bool;
      Bit_07_M199 : Bool;
      RecepOK_M200 : Bool;
      PresNormal_M200 : Bool;
      Ausencia_M200 : Bool;
      PresBloqueo_M200 : Bool;
      Galibo_M200 : Bool;
      PresPreparada_M200 : Bool;
      PresMultiple_M200 : Bool;
      Bit_07_M200 : Bool;
      RecepOK_M201 : Bool;
      PresNormal_M201 : Bool;
      Ausencia_M201 : Bool;
      PresBloqueo_M201 : Bool;
      Galibo_M201 : Bool;
      PresPreparada_M201 : Bool;
      PresMultiple_M201 : Bool;
      Bit_07_M201 : Bool;
      RecepOK_M202 : Bool;
      PresNormal_M202 : Bool;
      Ausencia_M202 : Bool;
      PresBloqueo_M202 : Bool;
      Galibo_M202 : Bool;
      PresPreparada_M202 : Bool;
      PresMultiple_M202 : Bool;
      Bit_07_M202 : Bool;
      RecepOK_M203 : Bool;
      PresNormal_M203 : Bool;
      Ausencia_M203 : Bool;
      PresBloqueo_M203 : Bool;
      Galibo_M203 : Bool;
      PresPreparada_M203 : Bool;
      PresMultiple_M203 : Bool;
      Bit_07_M203 : Bool;
      RecepOK_M204 : Bool;
      PresNormal_M204 : Bool;
      Ausencia_M204 : Bool;
      PresBloqueo_M204 : Bool;
      Galibo_M204 : Bool;
      PresPreparada_M204 : Bool;
      PresMultiple_M204 : Bool;
      Bit_07_M204 : Bool;
      RecepOK_M205 : Bool;
      PresNormal_M205 : Bool;
      Ausencia_M205 : Bool;
      PresBloqueo_M205 : Bool;
      Galibo_M205 : Bool;
      PresPreparada_M205 : Bool;
      PresMultiple_M205 : Bool;
      Bit_07_M205 : Bool;
      RecepOK_M206 : Bool;
      PresNormal_M206 : Bool;
      Ausencia_M206 : Bool;
      PresBloqueo_M206 : Bool;
      Galibo_M206 : Bool;
      PresPreparada_M206 : Bool;
      PresMultiple_M206 : Bool;
      Bit_07_M206 : Bool;
      RecepOK_M207 : Bool;
      PresNormal_M207 : Bool;
      Ausencia_M207 : Bool;
      PresBloqueo_M207 : Bool;
      Galibo_M207 : Bool;
      PresPreparada_M207 : Bool;
      PresMultiple_M207 : Bool;
      Bit_07_M207 : Bool;
      RecepOK_M208 : Bool;
      PresNormal_M208 : Bool;
      Ausencia_M208 : Bool;
      PresBloqueo_M208 : Bool;
      Galibo_M208 : Bool;
      PresPreparada_M208 : Bool;
      PresMultiple_M208 : Bool;
      Bit_07_M208 : Bool;
      RecepOK_M209 : Bool;
      PresNormal_M209 : Bool;
      Ausencia_M209 : Bool;
      PresBloqueo_M209 : Bool;
      Galibo_M209 : Bool;
      PresPreparada_M209 : Bool;
      PresMultiple_M209 : Bool;
      Bit_07_M209 : Bool;
      RecepOK_M210 : Bool;
      PresNormal_M210 : Bool;
      Ausencia_M210 : Bool;
      PresBloqueo_M210 : Bool;
      Galibo_M210 : Bool;
      PresPreparada_M210 : Bool;
      PresMultiple_M210 : Bool;
      Bit_07_M210 : Bool;
      RecepOK_M211 : Bool;
      PresNormal_M211 : Bool;
      Ausencia_M211 : Bool;
      PresBloqueo_M211 : Bool;
      Galibo_M211 : Bool;
      PresPreparada_M211 : Bool;
      PresMultiple_M211 : Bool;
      Bit_07_M211 : Bool;
      RecepOK_M212 : Bool;
      PresNormal_M212 : Bool;
      Ausencia_M212 : Bool;
      PresBloqueo_M212 : Bool;
      Galibo_M212 : Bool;
      PresPreparada_M212 : Bool;
      PresMultiple_M212 : Bool;
      Bit_07_M212 : Bool;
      RecepOK_M213 : Bool;
      PresNormal_M213 : Bool;
      Ausencia_M213 : Bool;
      PresBloqueo_M213 : Bool;
      Galibo_M213 : Bool;
      PresPreparada_M213 : Bool;
      PresMultiple_M213 : Bool;
      Bit_07_M213 : Bool;
      RecepOK_M214 : Bool;
      PresNormal_M214 : Bool;
      Ausencia_M214 : Bool;
      PresBloqueo_M214 : Bool;
      Galibo_M214 : Bool;
      PresPreparada_M214 : Bool;
      PresMultiple_M214 : Bool;
      Bit_07_M214 : Bool;
      RecepOK_M215 : Bool;
      PresNormal_M215 : Bool;
      Ausencia_M215 : Bool;
      PresBloqueo_M215 : Bool;
      Galibo_M215 : Bool;
      PresPreparada_M215 : Bool;
      PresMultiple_M215 : Bool;
      Bit_07_M215 : Bool;
      RecepOK_M216 : Bool;
      PresNormal_M216 : Bool;
      Ausencia_M216 : Bool;
      PresBloqueo_M216 : Bool;
      Galibo_M216 : Bool;
      PresPreparada_M216 : Bool;
      PresMultiple_M216 : Bool;
      Bit_07_M216 : Bool;
      RecepOK_M217 : Bool;
      PresNormal_M217 : Bool;
      Ausencia_M217 : Bool;
      PresBloqueo_M217 : Bool;
      Galibo_M217 : Bool;
      PresPreparada_M217 : Bool;
      PresMultiple_M217 : Bool;
      Bit_07_M217 : Bool;
      RecepOK_M218 : Bool;
      PresNormal_M218 : Bool;
      Ausencia_M218 : Bool;
      PresBloqueo_M218 : Bool;
      Galibo_M218 : Bool;
      PresPreparada_M218 : Bool;
      PresMultiple_M218 : Bool;
      Bit_07_M218 : Bool;
      RecepOK_M219 : Bool;
      PresNormal_M219 : Bool;
      Ausencia_M219 : Bool;
      PresBloqueo_M219 : Bool;
      Galibo_M219 : Bool;
      PresPreparada_M219 : Bool;
      PresMultiple_M219 : Bool;
      Bit_07_M219 : Bool;
      RecepOK_M220 : Bool;
      PresNormal_M220 : Bool;
      Ausencia_M220 : Bool;
      PresBloqueo_M220 : Bool;
      Galibo_M220 : Bool;
      PresPreparada_M220 : Bool;
      PresMultiple_M220 : Bool;
      Bit_07_M220 : Bool;
      RecepOK_M221 : Bool;
      PresNormal_M221 : Bool;
      Ausencia_M221 : Bool;
      PresBloqueo_M221 : Bool;
      Galibo_M221 : Bool;
      PresPreparada_M221 : Bool;
      PresMultiple_M221 : Bool;
      Bit_07_M221 : Bool;
      RecepOK_M222 : Bool;
      PresNormal_M222 : Bool;
      Ausencia_M222 : Bool;
      PresBloqueo_M222 : Bool;
      Galibo_M222 : Bool;
      PresPreparada_M222 : Bool;
      PresMultiple_M222 : Bool;
      Bit_07_M222 : Bool;
      RecepOK_M223 : Bool;
      PresNormal_M223 : Bool;
      Ausencia_M223 : Bool;
      PresBloqueo_M223 : Bool;
      Galibo_M223 : Bool;
      PresPreparada_M223 : Bool;
      PresMultiple_M223 : Bool;
      Bit_07_M223 : Bool;
      RecepOK_M224 : Bool;
      PresNormal_M224 : Bool;
      Ausencia_M224 : Bool;
      PresBloqueo_M224 : Bool;
      Galibo_M224 : Bool;
      PresPreparada_M224 : Bool;
      PresMultiple_M224 : Bool;
      Bit_07_M224 : Bool;
      RecepOK_M225 : Bool;
      PresNormal_M225 : Bool;
      Ausencia_M225 : Bool;
      PresBloqueo_M225 : Bool;
      Galibo_M225 : Bool;
      PresPreparada_M225 : Bool;
      PresMultiple_M225 : Bool;
      Bit_07_M225 : Bool;
      RecepOK_M226 : Bool;
      PresNormal_M226 : Bool;
      Ausencia_M226 : Bool;
      PresBloqueo_M226 : Bool;
      Galibo_M226 : Bool;
      PresPreparada_M226 : Bool;
      PresMultiple_M226 : Bool;
      Bit_07_M226 : Bool;
      RecepOK_M227 : Bool;
      PresNormal_M227 : Bool;
      Ausencia_M227 : Bool;
      PresBloqueo_M227 : Bool;
      Galibo_M227 : Bool;
      PresPreparada_M227 : Bool;
      PresMultiple_M227 : Bool;
      Bit_07_M227 : Bool;
      RecepOK_M228 : Bool;
      PresNormal_M228 : Bool;
      Ausencia_M228 : Bool;
      PresBloqueo_M228 : Bool;
      Galibo_M228 : Bool;
      PresPreparada_M228 : Bool;
      PresMultiple_M228 : Bool;
      Bit_07_M228 : Bool;
      RecepOK_M229 : Bool;
      PresNormal_M229 : Bool;
      Ausencia_M229 : Bool;
      PresBloqueo_M229 : Bool;
      Galibo_M229 : Bool;
      PresPreparada_M229 : Bool;
      PresMultiple_M229 : Bool;
      Bit_07_M229 : Bool;
      RecepOK_M230 : Bool;
      PresNormal_M230 : Bool;
      Ausencia_M230 : Bool;
      PresBloqueo_M230 : Bool;
      Galibo_M230 : Bool;
      PresPreparada_M230 : Bool;
      PresMultiple_M230 : Bool;
      Bit_07_M230 : Bool;
      RecepOK_M231 : Bool;
      PresNormal_M231 : Bool;
      Ausencia_M231 : Bool;
      PresBloqueo_M231 : Bool;
      Galibo_M231 : Bool;
      PresPreparada_M231 : Bool;
      PresMultiple_M231 : Bool;
      Bit_07_M231 : Bool;
      RecepOK_M232 : Bool;
      PresNormal_M232 : Bool;
      Ausencia_M232 : Bool;
      PresBloqueo_M232 : Bool;
      Galibo_M232 : Bool;
      PresPreparada_M232 : Bool;
      PresMultiple_M232 : Bool;
      Bit_07_M232 : Bool;
      RecepOK_M233 : Bool;
      PresNormal_M233 : Bool;
      Ausencia_M233 : Bool;
      PresBloqueo_M233 : Bool;
      Galibo_M233 : Bool;
      PresPreparada_M233 : Bool;
      PresMultiple_M233 : Bool;
      Bit_07_M233 : Bool;
      RecepOK_M234 : Bool;
      PresNormal_M234 : Bool;
      Ausencia_M234 : Bool;
      PresBloqueo_M234 : Bool;
      Galibo_M234 : Bool;
      PresPreparada_M234 : Bool;
      PresMultiple_M234 : Bool;
      Bit_07_M234 : Bool;
      RecepOK_M235 : Bool;
      PresNormal_M235 : Bool;
      Ausencia_M235 : Bool;
      PresBloqueo_M235 : Bool;
      Galibo_M235 : Bool;
      PresPreparada_M235 : Bool;
      PresMultiple_M235 : Bool;
      Bit_07_M235 : Bool;
      RecepOK_M236 : Bool;
      PresNormal_M236 : Bool;
      Ausencia_M236 : Bool;
      PresBloqueo_M236 : Bool;
      Galibo_M236 : Bool;
      PresPreparada_M236 : Bool;
      PresMultiple_M236 : Bool;
      Bit_07_M236 : Bool;
      RecepOK_M237 : Bool;
      PresNormal_M237 : Bool;
      Ausencia_M237 : Bool;
      PresBloqueo_M237 : Bool;
      Galibo_M237 : Bool;
      PresPreparada_M237 : Bool;
      PresMultiple_M237 : Bool;
      Bit_07_M237 : Bool;
      RecepOK_M238 : Bool;
      PresNormal_M238 : Bool;
      Ausencia_M238 : Bool;
      PresBloqueo_M238 : Bool;
      Galibo_M238 : Bool;
      PresPreparada_M238 : Bool;
      PresMultiple_M238 : Bool;
      Bit_07_M238 : Bool;
      RecepOK_M239 : Bool;
      PresNormal_M239 : Bool;
      Ausencia_M239 : Bool;
      PresBloqueo_M239 : Bool;
      Galibo_M239 : Bool;
      PresPreparada_M239 : Bool;
      PresMultiple_M239 : Bool;
      Bit_07_M239 : Bool;
      RecepOK_M240 : Bool;
      PresNormal_M240 : Bool;
      Ausencia_M240 : Bool;
      PresBloqueo_M240 : Bool;
      Galibo_M240 : Bool;
      PresPreparada_M240 : Bool;
      PresMultiple_M240 : Bool;
      Bit_07_M240 : Bool;
      RecepOK_M241 : Bool;
      PresNormal_M241 : Bool;
      Ausencia_M241 : Bool;
      PresBloqueo_M241 : Bool;
      Galibo_M241 : Bool;
      PresPreparada_M241 : Bool;
      PresMultiple_M241 : Bool;
      Bit_07_M241 : Bool;
      RecepOK_M242 : Bool;
      PresNormal_M242 : Bool;
      Ausencia_M242 : Bool;
      PresBloqueo_M242 : Bool;
      Galibo_M242 : Bool;
      PresPreparada_M242 : Bool;
      PresMultiple_M242 : Bool;
      Bit_07_M242 : Bool;
      RecepOK_M243 : Bool;
      PresNormal_M243 : Bool;
      Ausencia_M243 : Bool;
      PresBloqueo_M243 : Bool;
      Galibo_M243 : Bool;
      PresPreparada_M243 : Bool;
      PresMultiple_M243 : Bool;
      Bit_07_M243 : Bool;
      RecepOK_M244 : Bool;
      PresNormal_M244 : Bool;
      Ausencia_M244 : Bool;
      PresBloqueo_M244 : Bool;
      Galibo_M244 : Bool;
      PresPreparada_M244 : Bool;
      PresMultiple_M244 : Bool;
      Bit_07_M244 : Bool;
      RecepOK_M245 : Bool;
      PresNormal_M245 : Bool;
      Ausencia_M245 : Bool;
      PresBloqueo_M245 : Bool;
      Galibo_M245 : Bool;
      PresPreparada_M245 : Bool;
      PresMultiple_M245 : Bool;
      Bit_07_M245 : Bool;
      RecepOK_M246 : Bool;
      PresNormal_M246 : Bool;
      Ausencia_M246 : Bool;
      PresBloqueo_M246 : Bool;
      Galibo_M246 : Bool;
      PresPreparada_M246 : Bool;
      PresMultiple_M246 : Bool;
      Bit_07_M246 : Bool;
      RecepOK_M247 : Bool;
      PresNormal_M247 : Bool;
      Ausencia_M247 : Bool;
      PresBloqueo_M247 : Bool;
      Galibo_M247 : Bool;
      PresPreparada_M247 : Bool;
      PresMultiple_M247 : Bool;
      Bit_07_M247 : Bool;
      RecepOK_M248 : Bool;
      PresNormal_M248 : Bool;
      Ausencia_M248 : Bool;
      PresBloqueo_M248 : Bool;
      Galibo_M248 : Bool;
      PresPreparada_M248 : Bool;
      PresMultiple_M248 : Bool;
      Bit_07_M248 : Bool;
      RecepOK_M249 : Bool;
      PresNormal_M249 : Bool;
      Ausencia_M249 : Bool;
      PresBloqueo_M249 : Bool;
      Galibo_M249 : Bool;
      PresPreparada_M249 : Bool;
      PresMultiple_M249 : Bool;
      Bit_07_M249 : Bool;
      RecepOK_M250 : Bool;
      PresNormal_M250 : Bool;
      Ausencia_M250 : Bool;
      PresBloqueo_M250 : Bool;
      Galibo_M250 : Bool;
      PresPreparada_M250 : Bool;
      PresMultiple_M250 : Bool;
      Bit_07_M250 : Bool;
      RecepOK_M251 : Bool;
      PresNormal_M251 : Bool;
      Ausencia_M251 : Bool;
      PresBloqueo_M251 : Bool;
      Galibo_M251 : Bool;
      PresPreparada_M251 : Bool;
      PresMultiple_M251 : Bool;
      Bit_07_M251 : Bool;
      RecepOK_M252 : Bool;
      PresNormal_M252 : Bool;
      Ausencia_M252 : Bool;
      PresBloqueo_M252 : Bool;
      Galibo_M252 : Bool;
      PresPreparada_M252 : Bool;
      PresMultiple_M252 : Bool;
      Bit_07_M252 : Bool;
      RecepOK_M253 : Bool;
      PresNormal_M253 : Bool;
      Ausencia_M253 : Bool;
      PresBloqueo_M253 : Bool;
      Galibo_M253 : Bool;
      PresPreparada_M253 : Bool;
      PresMultiple_M253 : Bool;
      Bit_07_M253 : Bool;
      RecepOK_M254 : Bool;
      PresNormal_M254 : Bool;
      Ausencia_M254 : Bool;
      PresBloqueo_M254 : Bool;
      Galibo_M254 : Bool;
      PresPreparada_M254 : Bool;
      PresMultiple_M254 : Bool;
      Bit_07_M254 : Bool;
      RecepOK_M255 : Bool;
      PresNormal_M255 : Bool;
      Ausencia_M255 : Bool;
      PresBloqueo_M255 : Bool;
      Galibo_M255 : Bool;
      PresPreparada_M255 : Bool;
      PresMultiple_M255 : Bool;
      Bit_07_M255 : Bool;
      RecepOK_M256 : Bool;
      PresNormal_M256 : Bool;
      Ausencia_M256 : Bool;
      PresBloqueo_M256 : Bool;
      Galibo_M256 : Bool;
      PresPreparada_M256 : Bool;
      PresMultiple_M256 : Bool;
      Bit_07_M256 : Bool;
      RecepOK_M257 : Bool;
      PresNormal_M257 : Bool;
      Ausencia_M257 : Bool;
      PresBloqueo_M257 : Bool;
      Galibo_M257 : Bool;
      PresPreparada_M257 : Bool;
      PresMultiple_M257 : Bool;
      Bit_07_M257 : Bool;
      RecepOK_M258 : Bool;
      PresNormal_M258 : Bool;
      Ausencia_M258 : Bool;
      PresBloqueo_M258 : Bool;
      Galibo_M258 : Bool;
      PresPreparada_M258 : Bool;
      PresMultiple_M258 : Bool;
      Bit_07_M258 : Bool;
      RecepOK_M259 : Bool;
      PresNormal_M259 : Bool;
      Ausencia_M259 : Bool;
      PresBloqueo_M259 : Bool;
      Galibo_M259 : Bool;
      PresPreparada_M259 : Bool;
      PresMultiple_M259 : Bool;
      Bit_07_M259 : Bool;
      RecepOK_M260 : Bool;
      PresNormal_M260 : Bool;
      Ausencia_M260 : Bool;
      PresBloqueo_M260 : Bool;
      Galibo_M260 : Bool;
      PresPreparada_M260 : Bool;
      PresMultiple_M260 : Bool;
      Bit_07_M260 : Bool;
      RecepOK_M261 : Bool;
      PresNormal_M261 : Bool;
      Ausencia_M261 : Bool;
      PresBloqueo_M261 : Bool;
      Galibo_M261 : Bool;
      PresPreparada_M261 : Bool;
      PresMultiple_M261 : Bool;
      Bit_07_M261 : Bool;
      RecepOK_M262 : Bool;
      PresNormal_M262 : Bool;
      Ausencia_M262 : Bool;
      PresBloqueo_M262 : Bool;
      Galibo_M262 : Bool;
      PresPreparada_M262 : Bool;
      PresMultiple_M262 : Bool;
      Bit_07_M262 : Bool;
      RecepOK_M263 : Bool;
      PresNormal_M263 : Bool;
      Ausencia_M263 : Bool;
      PresBloqueo_M263 : Bool;
      Galibo_M263 : Bool;
      PresPreparada_M263 : Bool;
      PresMultiple_M263 : Bool;
      Bit_07_M263 : Bool;
      RecepOK_M264 : Bool;
      PresNormal_M264 : Bool;
      Ausencia_M264 : Bool;
      PresBloqueo_M264 : Bool;
      Galibo_M264 : Bool;
      PresPreparada_M264 : Bool;
      PresMultiple_M264 : Bool;
      Bit_07_M264 : Bool;
      RecepOK_M265 : Bool;
      PresNormal_M265 : Bool;
      Ausencia_M265 : Bool;
      PresBloqueo_M265 : Bool;
      Galibo_M265 : Bool;
      PresPreparada_M265 : Bool;
      PresMultiple_M265 : Bool;
      Bit_07_M265 : Bool;
      RecepOK_M266 : Bool;
      PresNormal_M266 : Bool;
      Ausencia_M266 : Bool;
      PresBloqueo_M266 : Bool;
      Galibo_M266 : Bool;
      PresPreparada_M266 : Bool;
      PresMultiple_M266 : Bool;
      Bit_07_M266 : Bool;
      RecepOK_M267 : Bool;
      PresNormal_M267 : Bool;
      Ausencia_M267 : Bool;
      PresBloqueo_M267 : Bool;
      Galibo_M267 : Bool;
      PresPreparada_M267 : Bool;
      PresMultiple_M267 : Bool;
      Bit_07_M267 : Bool;
      RecepOK_M268 : Bool;
      PresNormal_M268 : Bool;
      Ausencia_M268 : Bool;
      PresBloqueo_M268 : Bool;
      Galibo_M268 : Bool;
      PresPreparada_M268 : Bool;
      PresMultiple_M268 : Bool;
      Bit_07_M268 : Bool;
      RecepOK_M269 : Bool;
      PresNormal_M269 : Bool;
      Ausencia_M269 : Bool;
      PresBloqueo_M269 : Bool;
      Galibo_M269 : Bool;
      PresPreparada_M269 : Bool;
      PresMultiple_M269 : Bool;
      Bit_07_M269 : Bool;
      RecepOK_M270 : Bool;
      PresNormal_M270 : Bool;
      Ausencia_M270 : Bool;
      PresBloqueo_M270 : Bool;
      Galibo_M270 : Bool;
      PresPreparada_M270 : Bool;
      PresMultiple_M270 : Bool;
      Bit_07_M270 : Bool;
      RecepOK_M271 : Bool;
      PresNormal_M271 : Bool;
      Ausencia_M271 : Bool;
      PresBloqueo_M271 : Bool;
      Galibo_M271 : Bool;
      PresPreparada_M271 : Bool;
      PresMultiple_M271 : Bool;
      Bit_07_M271 : Bool;
      RecepOK_M272 : Bool;
      PresNormal_M272 : Bool;
      Ausencia_M272 : Bool;
      PresBloqueo_M272 : Bool;
      Galibo_M272 : Bool;
      PresPreparada_M272 : Bool;
      PresMultiple_M272 : Bool;
      Bit_07_M272 : Bool;
      RecepOK_M273 : Bool;
      PresNormal_M273 : Bool;
      Ausencia_M273 : Bool;
      PresBloqueo_M273 : Bool;
      Galibo_M273 : Bool;
      PresPreparada_M273 : Bool;
      PresMultiple_M273 : Bool;
      Bit_07_M273 : Bool;
      RecepOK_M274 : Bool;
      PresNormal_M274 : Bool;
      Ausencia_M274 : Bool;
      PresBloqueo_M274 : Bool;
      Galibo_M274 : Bool;
      PresPreparada_M274 : Bool;
      PresMultiple_M274 : Bool;
      Bit_07_M274 : Bool;
      RecepOK_M275 : Bool;
      PresNormal_M275 : Bool;
      Ausencia_M275 : Bool;
      PresBloqueo_M275 : Bool;
      Galibo_M275 : Bool;
      PresPreparada_M275 : Bool;
      PresMultiple_M275 : Bool;
      Bit_07_M275 : Bool;
      RecepOK_M276 : Bool;
      PresNormal_M276 : Bool;
      Ausencia_M276 : Bool;
      PresBloqueo_M276 : Bool;
      Galibo_M276 : Bool;
      PresPreparada_M276 : Bool;
      PresMultiple_M276 : Bool;
      Bit_07_M276 : Bool;
      RecepOK_M277 : Bool;
      PresNormal_M277 : Bool;
      Ausencia_M277 : Bool;
      PresBloqueo_M277 : Bool;
      Galibo_M277 : Bool;
      PresPreparada_M277 : Bool;
      PresMultiple_M277 : Bool;
      Bit_07_M277 : Bool;
      RecepOK_M278 : Bool;
      PresNormal_M278 : Bool;
      Ausencia_M278 : Bool;
      PresBloqueo_M278 : Bool;
      Galibo_M278 : Bool;
      PresPreparada_M278 : Bool;
      PresMultiple_M278 : Bool;
      Bit_07_M278 : Bool;
      RecepOK_M279 : Bool;
      PresNormal_M279 : Bool;
      Ausencia_M279 : Bool;
      PresBloqueo_M279 : Bool;
      Galibo_M279 : Bool;
      PresPreparada_M279 : Bool;
      PresMultiple_M279 : Bool;
      Bit_07_M279 : Bool;
      RecepOK_M280 : Bool;
      PresNormal_M280 : Bool;
      Ausencia_M280 : Bool;
      PresBloqueo_M280 : Bool;
      Galibo_M280 : Bool;
      PresPreparada_M280 : Bool;
      PresMultiple_M280 : Bool;
      Bit_07_M280 : Bool;
      RecepOK_M281 : Bool;
      PresNormal_M281 : Bool;
      Ausencia_M281 : Bool;
      PresBloqueo_M281 : Bool;
      Galibo_M281 : Bool;
      PresPreparada_M281 : Bool;
      PresMultiple_M281 : Bool;
      Bit_07_M281 : Bool;
      RecepOK_M282 : Bool;
      PresNormal_M282 : Bool;
      Ausencia_M282 : Bool;
      PresBloqueo_M282 : Bool;
      Galibo_M282 : Bool;
      PresPreparada_M282 : Bool;
      PresMultiple_M282 : Bool;
      Bit_07_M282 : Bool;
      RecepOK_M283 : Bool;
      PresNormal_M283 : Bool;
      Ausencia_M283 : Bool;
      PresBloqueo_M283 : Bool;
      Galibo_M283 : Bool;
      PresPreparada_M283 : Bool;
      PresMultiple_M283 : Bool;
      Bit_07_M283 : Bool;
      RecepOK_M284 : Bool;
      PresNormal_M284 : Bool;
      Ausencia_M284 : Bool;
      PresBloqueo_M284 : Bool;
      Galibo_M284 : Bool;
      PresPreparada_M284 : Bool;
      PresMultiple_M284 : Bool;
      Bit_07_M284 : Bool;
      RecepOK_M285 : Bool;
      PresNormal_M285 : Bool;
      Ausencia_M285 : Bool;
      PresBloqueo_M285 : Bool;
      Galibo_M285 : Bool;
      PresPreparada_M285 : Bool;
      PresMultiple_M285 : Bool;
      Bit_07_M285 : Bool;
      RecepOK_M286 : Bool;
      PresNormal_M286 : Bool;
      Ausencia_M286 : Bool;
      PresBloqueo_M286 : Bool;
      Galibo_M286 : Bool;
      PresPreparada_M286 : Bool;
      PresMultiple_M286 : Bool;
      Bit_07_M286 : Bool;
      RecepOK_M287 : Bool;
      PresNormal_M287 : Bool;
      Ausencia_M287 : Bool;
      PresBloqueo_M287 : Bool;
      Galibo_M287 : Bool;
      PresPreparada_M287 : Bool;
      PresMultiple_M287 : Bool;
      Bit_07_M287 : Bool;
      RecepOK_M288 : Bool;
      PresNormal_M288 : Bool;
      Ausencia_M288 : Bool;
      PresBloqueo_M288 : Bool;
      Galibo_M288 : Bool;
      PresPreparada_M288 : Bool;
      PresMultiple_M288 : Bool;
      Bit_07_M288 : Bool;
      RecepOK_M289 : Bool;
      PresNormal_M289 : Bool;
      Ausencia_M289 : Bool;
      PresBloqueo_M289 : Bool;
      Galibo_M289 : Bool;
      PresPreparada_M289 : Bool;
      PresMultiple_M289 : Bool;
      Bit_07_M289 : Bool;
      RecepOK_M290 : Bool;
      PresNormal_M290 : Bool;
      Ausencia_M290 : Bool;
      PresBloqueo_M290 : Bool;
      Galibo_M290 : Bool;
      PresPreparada_M290 : Bool;
      PresMultiple_M290 : Bool;
      Bit_07_M290 : Bool;
      RecepOK_M291 : Bool;
      PresNormal_M291 : Bool;
      Ausencia_M291 : Bool;
      PresBloqueo_M291 : Bool;
      Galibo_M291 : Bool;
      PresPreparada_M291 : Bool;
      PresMultiple_M291 : Bool;
      Bit_07_M291 : Bool;
      RecepOK_M292 : Bool;
      PresNormal_M292 : Bool;
      Ausencia_M292 : Bool;
      PresBloqueo_M292 : Bool;
      Galibo_M292 : Bool;
      PresPreparada_M292 : Bool;
      PresMultiple_M292 : Bool;
      Bit_07_M292 : Bool;
      RecepOK_M293 : Bool;
      PresNormal_M293 : Bool;
      Ausencia_M293 : Bool;
      PresBloqueo_M293 : Bool;
      Galibo_M293 : Bool;
      PresPreparada_M293 : Bool;
      PresMultiple_M293 : Bool;
      Bit_07_M293 : Bool;
      RecepOK_M294 : Bool;
      PresNormal_M294 : Bool;
      Ausencia_M294 : Bool;
      PresBloqueo_M294 : Bool;
      Galibo_M294 : Bool;
      PresPreparada_M294 : Bool;
      PresMultiple_M294 : Bool;
      Bit_07_M294 : Bool;
      RecepOK_M295 : Bool;
      PresNormal_M295 : Bool;
      Ausencia_M295 : Bool;
      PresBloqueo_M295 : Bool;
      Galibo_M295 : Bool;
      PresPreparada_M295 : Bool;
      PresMultiple_M295 : Bool;
      Bit_07_M295 : Bool;
      RecepOK_M296 : Bool;
      PresNormal_M296 : Bool;
      Ausencia_M296 : Bool;
      PresBloqueo_M296 : Bool;
      Galibo_M296 : Bool;
      PresPreparada_M296 : Bool;
      PresMultiple_M296 : Bool;
      Bit_07_M296 : Bool;
      RecepOK_M297 : Bool;
      PresNormal_M297 : Bool;
      Ausencia_M297 : Bool;
      PresBloqueo_M297 : Bool;
      Galibo_M297 : Bool;
      PresPreparada_M297 : Bool;
      PresMultiple_M297 : Bool;
      Bit_07_M297 : Bool;
      RecepOK_M298 : Bool;
      PresNormal_M298 : Bool;
      Ausencia_M298 : Bool;
      PresBloqueo_M298 : Bool;
      Galibo_M298 : Bool;
      PresPreparada_M298 : Bool;
      PresMultiple_M298 : Bool;
      Bit_07_M298 : Bool;
      RecepOK_M299 : Bool;
      PresNormal_M299 : Bool;
      Ausencia_M299 : Bool;
      PresBloqueo_M299 : Bool;
      Galibo_M299 : Bool;
      PresPreparada_M299 : Bool;
      PresMultiple_M299 : Bool;
      Bit_07_M299 : Bool;
      RecepOK_M300 : Bool;
      PresNormal_M300 : Bool;
      Ausencia_M300 : Bool;
      PresBloqueo_M300 : Bool;
      Galibo_M300 : Bool;
      PresPreparada_M300 : Bool;
      PresMultiple_M300 : Bool;
      Bit_07_M300 : Bool;
      RecepOK_M301 : Bool;
      PresNormal_M301 : Bool;
      Ausencia_M301 : Bool;
      PresBloqueo_M301 : Bool;
      Galibo_M301 : Bool;
      PresPreparada_M301 : Bool;
      PresMultiple_M301 : Bool;
      Bit_07_M301 : Bool;
      RecepOK_M302 : Bool;
      PresNormal_M302 : Bool;
      Ausencia_M302 : Bool;
      PresBloqueo_M302 : Bool;
      Galibo_M302 : Bool;
      PresPreparada_M302 : Bool;
      PresMultiple_M302 : Bool;
      Bit_07_M302 : Bool;
      RecepOK_M303 : Bool;
      PresNormal_M303 : Bool;
      Ausencia_M303 : Bool;
      PresBloqueo_M303 : Bool;
      Galibo_M303 : Bool;
      PresPreparada_M303 : Bool;
      PresMultiple_M303 : Bool;
      Bit_07_M303 : Bool;
      RecepOK_M304 : Bool;
      PresNormal_M304 : Bool;
      Ausencia_M304 : Bool;
      PresBloqueo_M304 : Bool;
      Galibo_M304 : Bool;
      PresPreparada_M304 : Bool;
      PresMultiple_M304 : Bool;
      Bit_07_M304 : Bool;
      RecepOK_M305 : Bool;
      PresNormal_M305 : Bool;
      Ausencia_M305 : Bool;
      PresBloqueo_M305 : Bool;
      Galibo_M305 : Bool;
      PresPreparada_M305 : Bool;
      PresMultiple_M305 : Bool;
      Bit_07_M305 : Bool;
      RecepOK_M306 : Bool;
      PresNormal_M306 : Bool;
      Ausencia_M306 : Bool;
      PresBloqueo_M306 : Bool;
      Galibo_M306 : Bool;
      PresPreparada_M306 : Bool;
      PresMultiple_M306 : Bool;
      Bit_07_M306 : Bool;
      RecepOK_M307 : Bool;
      PresNormal_M307 : Bool;
      Ausencia_M307 : Bool;
      PresBloqueo_M307 : Bool;
      Galibo_M307 : Bool;
      PresPreparada_M307 : Bool;
      PresMultiple_M307 : Bool;
      Bit_07_M307 : Bool;
      RecepOK_M308 : Bool;
      PresNormal_M308 : Bool;
      Ausencia_M308 : Bool;
      PresBloqueo_M308 : Bool;
      Galibo_M308 : Bool;
      PresPreparada_M308 : Bool;
      PresMultiple_M308 : Bool;
      Bit_07_M308 : Bool;
      RecepOK_M309 : Bool;
      PresNormal_M309 : Bool;
      Ausencia_M309 : Bool;
      PresBloqueo_M309 : Bool;
      Galibo_M309 : Bool;
      PresPreparada_M309 : Bool;
      PresMultiple_M309 : Bool;
      Bit_07_M309 : Bool;
      RecepOK_M310 : Bool;
      PresNormal_M310 : Bool;
      Ausencia_M310 : Bool;
      PresBloqueo_M310 : Bool;
      Galibo_M310 : Bool;
      PresPreparada_M310 : Bool;
      PresMultiple_M310 : Bool;
      Bit_07_M310 : Bool;
      RecepOK_M311 : Bool;
      PresNormal_M311 : Bool;
      Ausencia_M311 : Bool;
      PresBloqueo_M311 : Bool;
      Galibo_M311 : Bool;
      PresPreparada_M311 : Bool;
      PresMultiple_M311 : Bool;
      Bit_07_M311 : Bool;
      RecepOK_M312 : Bool;
      PresNormal_M312 : Bool;
      Ausencia_M312 : Bool;
      PresBloqueo_M312 : Bool;
      Galibo_M312 : Bool;
      PresPreparada_M312 : Bool;
      PresMultiple_M312 : Bool;
      Bit_07_M312 : Bool;
      RecepOK_M313 : Bool;
      PresNormal_M313 : Bool;
      Ausencia_M313 : Bool;
      PresBloqueo_M313 : Bool;
      Galibo_M313 : Bool;
      PresPreparada_M313 : Bool;
      PresMultiple_M313 : Bool;
      Bit_07_M313 : Bool;
      RecepOK_M314 : Bool;
      PresNormal_M314 : Bool;
      Ausencia_M314 : Bool;
      PresBloqueo_M314 : Bool;
      Galibo_M314 : Bool;
      PresPreparada_M314 : Bool;
      PresMultiple_M314 : Bool;
      Bit_07_M314 : Bool;
      RecepOK_M315 : Bool;
      PresNormal_M315 : Bool;
      Ausencia_M315 : Bool;
      PresBloqueo_M315 : Bool;
      Galibo_M315 : Bool;
      PresPreparada_M315 : Bool;
      PresMultiple_M315 : Bool;
      Bit_07_M315 : Bool;
      RecepOK_M316 : Bool;
      PresNormal_M316 : Bool;
      Ausencia_M316 : Bool;
      PresBloqueo_M316 : Bool;
      Galibo_M316 : Bool;
      PresPreparada_M316 : Bool;
      PresMultiple_M316 : Bool;
      Bit_07_M316 : Bool;
      RecepOK_M317 : Bool;
      PresNormal_M317 : Bool;
      Ausencia_M317 : Bool;
      PresBloqueo_M317 : Bool;
      Galibo_M317 : Bool;
      PresPreparada_M317 : Bool;
      PresMultiple_M317 : Bool;
      Bit_07_M317 : Bool;
      RecepOK_M318 : Bool;
      PresNormal_M318 : Bool;
      Ausencia_M318 : Bool;
      PresBloqueo_M318 : Bool;
      Galibo_M318 : Bool;
      PresPreparada_M318 : Bool;
      PresMultiple_M318 : Bool;
      Bit_07_M318 : Bool;
      RecepOK_M319 : Bool;
      PresNormal_M319 : Bool;
      Ausencia_M319 : Bool;
      PresBloqueo_M319 : Bool;
      Galibo_M319 : Bool;
      PresPreparada_M319 : Bool;
      PresMultiple_M319 : Bool;
      Bit_07_M319 : Bool;
      RecepOK_M320 : Bool;
      PresNormal_M320 : Bool;
      Ausencia_M320 : Bool;
      PresBloqueo_M320 : Bool;
      Galibo_M320 : Bool;
      PresPreparada_M320 : Bool;
      PresMultiple_M320 : Bool;
      Bit_07_M320 : Bool;
      RecepOK_M321 : Bool;
      PresNormal_M321 : Bool;
      Ausencia_M321 : Bool;
      PresBloqueo_M321 : Bool;
      Galibo_M321 : Bool;
      PresPreparada_M321 : Bool;
      PresMultiple_M321 : Bool;
      Bit_07_M321 : Bool;
      RecepOK_M322 : Bool;
      PresNormal_M322 : Bool;
      Ausencia_M322 : Bool;
      PresBloqueo_M322 : Bool;
      Galibo_M322 : Bool;
      PresPreparada_M322 : Bool;
      PresMultiple_M322 : Bool;
      Bit_07_M322 : Bool;
      RecepOK_M323 : Bool;
      PresNormal_M323 : Bool;
      Ausencia_M323 : Bool;
      PresBloqueo_M323 : Bool;
      Galibo_M323 : Bool;
      PresPreparada_M323 : Bool;
      PresMultiple_M323 : Bool;
      Bit_07_M323 : Bool;
      RecepOK_M324 : Bool;
      PresNormal_M324 : Bool;
      Ausencia_M324 : Bool;
      PresBloqueo_M324 : Bool;
      Galibo_M324 : Bool;
      PresPreparada_M324 : Bool;
      PresMultiple_M324 : Bool;
      Bit_07_M324 : Bool;
      RecepOK_M325 : Bool;
      PresNormal_M325 : Bool;
      Ausencia_M325 : Bool;
      PresBloqueo_M325 : Bool;
      Galibo_M325 : Bool;
      PresPreparada_M325 : Bool;
      PresMultiple_M325 : Bool;
      Bit_07_M325 : Bool;
      RecepOK_M326 : Bool;
      PresNormal_M326 : Bool;
      Ausencia_M326 : Bool;
      PresBloqueo_M326 : Bool;
      Galibo_M326 : Bool;
      PresPreparada_M326 : Bool;
      PresMultiple_M326 : Bool;
      Bit_07_M326 : Bool;
      RecepOK_M327 : Bool;
      PresNormal_M327 : Bool;
      Ausencia_M327 : Bool;
      PresBloqueo_M327 : Bool;
      Galibo_M327 : Bool;
      PresPreparada_M327 : Bool;
      PresMultiple_M327 : Bool;
      Bit_07_M327 : Bool;
      RecepOK_M328 : Bool;
      PresNormal_M328 : Bool;
      Ausencia_M328 : Bool;
      PresBloqueo_M328 : Bool;
      Galibo_M328 : Bool;
      PresPreparada_M328 : Bool;
      PresMultiple_M328 : Bool;
      Bit_07_M328 : Bool;
      RecepOK_M329 : Bool;
      PresNormal_M329 : Bool;
      Ausencia_M329 : Bool;
      PresBloqueo_M329 : Bool;
      Galibo_M329 : Bool;
      PresPreparada_M329 : Bool;
      PresMultiple_M329 : Bool;
      Bit_07_M329 : Bool;
      RecepOK_M330 : Bool;
      PresNormal_M330 : Bool;
      Ausencia_M330 : Bool;
      PresBloqueo_M330 : Bool;
      Galibo_M330 : Bool;
      PresPreparada_M330 : Bool;
      PresMultiple_M330 : Bool;
      Bit_07_M330 : Bool;
      RecepOK_M331 : Bool;
      PresNormal_M331 : Bool;
      Ausencia_M331 : Bool;
      PresBloqueo_M331 : Bool;
      Galibo_M331 : Bool;
      PresPreparada_M331 : Bool;
      PresMultiple_M331 : Bool;
      Bit_07_M331 : Bool;
      RecepOK_M332 : Bool;
      PresNormal_M332 : Bool;
      Ausencia_M332 : Bool;
      PresBloqueo_M332 : Bool;
      Galibo_M332 : Bool;
      PresPreparada_M332 : Bool;
      PresMultiple_M332 : Bool;
      Bit_07_M332 : Bool;
      RecepOK_M333 : Bool;
      PresNormal_M333 : Bool;
      Ausencia_M333 : Bool;
      PresBloqueo_M333 : Bool;
      Galibo_M333 : Bool;
      PresPreparada_M333 : Bool;
      PresMultiple_M333 : Bool;
      Bit_07_M333 : Bool;
      RecepOK_M334 : Bool;
      PresNormal_M334 : Bool;
      Ausencia_M334 : Bool;
      PresBloqueo_M334 : Bool;
      Galibo_M334 : Bool;
      PresPreparada_M334 : Bool;
      PresMultiple_M334 : Bool;
      Bit_07_M334 : Bool;
      RecepOK_M335 : Bool;
      PresNormal_M335 : Bool;
      Ausencia_M335 : Bool;
      PresBloqueo_M335 : Bool;
      Galibo_M335 : Bool;
      PresPreparada_M335 : Bool;
      PresMultiple_M335 : Bool;
      Bit_07_M335 : Bool;
      RecepOK_M336 : Bool;
      PresNormal_M336 : Bool;
      Ausencia_M336 : Bool;
      PresBloqueo_M336 : Bool;
      Galibo_M336 : Bool;
      PresPreparada_M336 : Bool;
      PresMultiple_M336 : Bool;
      Bit_07_M336 : Bool;
      RecepOK_M337 : Bool;
      PresNormal_M337 : Bool;
      Ausencia_M337 : Bool;
      PresBloqueo_M337 : Bool;
      Galibo_M337 : Bool;
      PresPreparada_M337 : Bool;
      PresMultiple_M337 : Bool;
      Bit_07_M337 : Bool;
      RecepOK_M338 : Bool;
      PresNormal_M338 : Bool;
      Ausencia_M338 : Bool;
      PresBloqueo_M338 : Bool;
      Galibo_M338 : Bool;
      PresPreparada_M338 : Bool;
      PresMultiple_M338 : Bool;
      Bit_07_M338 : Bool;
      RecepOK_M339 : Bool;
      PresNormal_M339 : Bool;
      Ausencia_M339 : Bool;
      PresBloqueo_M339 : Bool;
      Galibo_M339 : Bool;
      PresPreparada_M339 : Bool;
      PresMultiple_M339 : Bool;
      Bit_07_M339 : Bool;
      RecepOK_M340 : Bool;
      PresNormal_M340 : Bool;
      Ausencia_M340 : Bool;
      PresBloqueo_M340 : Bool;
      Galibo_M340 : Bool;
      PresPreparada_M340 : Bool;
      PresMultiple_M340 : Bool;
      Bit_07_M340 : Bool;
      RecepOK_M341 : Bool;
      PresNormal_M341 : Bool;
      Ausencia_M341 : Bool;
      PresBloqueo_M341 : Bool;
      Galibo_M341 : Bool;
      PresPreparada_M341 : Bool;
      PresMultiple_M341 : Bool;
      Bit_07_M341 : Bool;
      RecepOK_M342 : Bool;
      PresNormal_M342 : Bool;
      Ausencia_M342 : Bool;
      PresBloqueo_M342 : Bool;
      Galibo_M342 : Bool;
      PresPreparada_M342 : Bool;
      PresMultiple_M342 : Bool;
      Bit_07_M342 : Bool;
      RecepOK_M343 : Bool;
      PresNormal_M343 : Bool;
      Ausencia_M343 : Bool;
      PresBloqueo_M343 : Bool;
      Galibo_M343 : Bool;
      PresPreparada_M343 : Bool;
      PresMultiple_M343 : Bool;
      Bit_07_M343 : Bool;
      RecepOK_M344 : Bool;
      PresNormal_M344 : Bool;
      Ausencia_M344 : Bool;
      PresBloqueo_M344 : Bool;
      Galibo_M344 : Bool;
      PresPreparada_M344 : Bool;
      PresMultiple_M344 : Bool;
      Bit_07_M344 : Bool;
      RecepOK_M345 : Bool;
      PresNormal_M345 : Bool;
      Ausencia_M345 : Bool;
      PresBloqueo_M345 : Bool;
      Galibo_M345 : Bool;
      PresPreparada_M345 : Bool;
      PresMultiple_M345 : Bool;
      Bit_07_M345 : Bool;
      RecepOK_M346 : Bool;
      PresNormal_M346 : Bool;
      Ausencia_M346 : Bool;
      PresBloqueo_M346 : Bool;
      Galibo_M346 : Bool;
      PresPreparada_M346 : Bool;
      PresMultiple_M346 : Bool;
      Bit_07_M346 : Bool;
      RecepOK_M347 : Bool;
      PresNormal_M347 : Bool;
      Ausencia_M347 : Bool;
      PresBloqueo_M347 : Bool;
      Galibo_M347 : Bool;
      PresPreparada_M347 : Bool;
      PresMultiple_M347 : Bool;
      Bit_07_M347 : Bool;
      RecepOK_M348 : Bool;
      PresNormal_M348 : Bool;
      Ausencia_M348 : Bool;
      PresBloqueo_M348 : Bool;
      Galibo_M348 : Bool;
      PresPreparada_M348 : Bool;
      PresMultiple_M348 : Bool;
      Bit_07_M348 : Bool;
      RecepOK_M349 : Bool;
      PresNormal_M349 : Bool;
      Ausencia_M349 : Bool;
      PresBloqueo_M349 : Bool;
      Galibo_M349 : Bool;
      PresPreparada_M349 : Bool;
      PresMultiple_M349 : Bool;
      Bit_07_M349 : Bool;
      RecepOK_M350 : Bool;
      PresNormal_M350 : Bool;
      Ausencia_M350 : Bool;
      PresBloqueo_M350 : Bool;
      Galibo_M350 : Bool;
      PresPreparada_M350 : Bool;
      PresMultiple_M350 : Bool;
      Bit_07_M350 : Bool;
      RecepOK_M351 : Bool;
      PresNormal_M351 : Bool;
      Ausencia_M351 : Bool;
      PresBloqueo_M351 : Bool;
      Galibo_M351 : Bool;
      PresPreparada_M351 : Bool;
      PresMultiple_M351 : Bool;
      Bit_07_M351 : Bool;
      RecepOK_M352 : Bool;
      PresNormal_M352 : Bool;
      Ausencia_M352 : Bool;
      PresBloqueo_M352 : Bool;
      Galibo_M352 : Bool;
      PresPreparada_M352 : Bool;
      PresMultiple_M352 : Bool;
      Bit_07_M352 : Bool;
      RecepOK_M353 : Bool;
      PresNormal_M353 : Bool;
      Ausencia_M353 : Bool;
      PresBloqueo_M353 : Bool;
      Galibo_M353 : Bool;
      PresPreparada_M353 : Bool;
      PresMultiple_M353 : Bool;
      Bit_07_M353 : Bool;
      RecepOK_M354 : Bool;
      PresNormal_M354 : Bool;
      Ausencia_M354 : Bool;
      PresBloqueo_M354 : Bool;
      Galibo_M354 : Bool;
      PresPreparada_M354 : Bool;
      PresMultiple_M354 : Bool;
      Bit_07_M354 : Bool;
      RecepOK_M355 : Bool;
      PresNormal_M355 : Bool;
      Ausencia_M355 : Bool;
      PresBloqueo_M355 : Bool;
      Galibo_M355 : Bool;
      PresPreparada_M355 : Bool;
      PresMultiple_M355 : Bool;
      Bit_07_M355 : Bool;
      RecepOK_M356 : Bool;
      PresNormal_M356 : Bool;
      Ausencia_M356 : Bool;
      PresBloqueo_M356 : Bool;
      Galibo_M356 : Bool;
      PresPreparada_M356 : Bool;
      PresMultiple_M356 : Bool;
      Bit_07_M356 : Bool;
      RecepOK_M357 : Bool;
      PresNormal_M357 : Bool;
      Ausencia_M357 : Bool;
      PresBloqueo_M357 : Bool;
      Galibo_M357 : Bool;
      PresPreparada_M357 : Bool;
      PresMultiple_M357 : Bool;
      Bit_07_M357 : Bool;
      RecepOK_M358 : Bool;
      PresNormal_M358 : Bool;
      Ausencia_M358 : Bool;
      PresBloqueo_M358 : Bool;
      Galibo_M358 : Bool;
      PresPreparada_M358 : Bool;
      PresMultiple_M358 : Bool;
      Bit_07_M358 : Bool;
      RecepOK_M359 : Bool;
      PresNormal_M359 : Bool;
      Ausencia_M359 : Bool;
      PresBloqueo_M359 : Bool;
      Galibo_M359 : Bool;
      PresPreparada_M359 : Bool;
      PresMultiple_M359 : Bool;
      Bit_07_M359 : Bool;
      RecepOK_M360 : Bool;
      PresNormal_M360 : Bool;
      Ausencia_M360 : Bool;
      PresBloqueo_M360 : Bool;
      Galibo_M360 : Bool;
      PresPreparada_M360 : Bool;
      PresMultiple_M360 : Bool;
      Bit_07_M360 : Bool;
      RecepOK_M361 : Bool;
      PresNormal_M361 : Bool;
      Ausencia_M361 : Bool;
      PresBloqueo_M361 : Bool;
      Galibo_M361 : Bool;
      PresPreparada_M361 : Bool;
      PresMultiple_M361 : Bool;
      Bit_07_M361 : Bool;
      RecepOK_M362 : Bool;
      PresNormal_M362 : Bool;
      Ausencia_M362 : Bool;
      PresBloqueo_M362 : Bool;
      Galibo_M362 : Bool;
      PresPreparada_M362 : Bool;
      PresMultiple_M362 : Bool;
      Bit_07_M362 : Bool;
      RecepOK_M363 : Bool;
      PresNormal_M363 : Bool;
      Ausencia_M363 : Bool;
      PresBloqueo_M363 : Bool;
      Galibo_M363 : Bool;
      PresPreparada_M363 : Bool;
      PresMultiple_M363 : Bool;
      Bit_07_M363 : Bool;
      RecepOK_M364 : Bool;
      PresNormal_M364 : Bool;
      Ausencia_M364 : Bool;
      PresBloqueo_M364 : Bool;
      Galibo_M364 : Bool;
      PresPreparada_M364 : Bool;
      PresMultiple_M364 : Bool;
      Bit_07_M364 : Bool;
      RecepOK_M365 : Bool;
      PresNormal_M365 : Bool;
      Ausencia_M365 : Bool;
      PresBloqueo_M365 : Bool;
      Galibo_M365 : Bool;
      PresPreparada_M365 : Bool;
      PresMultiple_M365 : Bool;
      Bit_07_M365 : Bool;
      RecepOK_M366 : Bool;
      PresNormal_M366 : Bool;
      Ausencia_M366 : Bool;
      PresBloqueo_M366 : Bool;
      Galibo_M366 : Bool;
      PresPreparada_M366 : Bool;
      PresMultiple_M366 : Bool;
      Bit_07_M366 : Bool;
      RecepOK_M367 : Bool;
      PresNormal_M367 : Bool;
      Ausencia_M367 : Bool;
      PresBloqueo_M367 : Bool;
      Galibo_M367 : Bool;
      PresPreparada_M367 : Bool;
      PresMultiple_M367 : Bool;
      Bit_07_M367 : Bool;
      RecepOK_M368 : Bool;
      PresNormal_M368 : Bool;
      Ausencia_M368 : Bool;
      PresBloqueo_M368 : Bool;
      Galibo_M368 : Bool;
      PresPreparada_M368 : Bool;
      PresMultiple_M368 : Bool;
      Bit_07_M368 : Bool;
      RecepOK_M369 : Bool;
      PresNormal_M369 : Bool;
      Ausencia_M369 : Bool;
      PresBloqueo_M369 : Bool;
      Galibo_M369 : Bool;
      PresPreparada_M369 : Bool;
      PresMultiple_M369 : Bool;
      Bit_07_M369 : Bool;
      RecepOK_M370 : Bool;
      PresNormal_M370 : Bool;
      Ausencia_M370 : Bool;
      PresBloqueo_M370 : Bool;
      Galibo_M370 : Bool;
      PresPreparada_M370 : Bool;
      PresMultiple_M370 : Bool;
      Bit_07_M370 : Bool;
      RecepOK_M371 : Bool;
      PresNormal_M371 : Bool;
      Ausencia_M371 : Bool;
      PresBloqueo_M371 : Bool;
      Galibo_M371 : Bool;
      PresPreparada_M371 : Bool;
      PresMultiple_M371 : Bool;
      Bit_07_M371 : Bool;
      RecepOK_M372 : Bool;
      PresNormal_M372 : Bool;
      Ausencia_M372 : Bool;
      PresBloqueo_M372 : Bool;
      Galibo_M372 : Bool;
      PresPreparada_M372 : Bool;
      PresMultiple_M372 : Bool;
      Bit_07_M372 : Bool;
      RecepOK_M373 : Bool;
      PresNormal_M373 : Bool;
      Ausencia_M373 : Bool;
      PresBloqueo_M373 : Bool;
      Galibo_M373 : Bool;
      PresPreparada_M373 : Bool;
      PresMultiple_M373 : Bool;
      Bit_07_M373 : Bool;
      RecepOK_M374 : Bool;
      PresNormal_M374 : Bool;
      Ausencia_M374 : Bool;
      PresBloqueo_M374 : Bool;
      Galibo_M374 : Bool;
      PresPreparada_M374 : Bool;
      PresMultiple_M374 : Bool;
      Bit_07_M374 : Bool;
      RecepOK_M375 : Bool;
      PresNormal_M375 : Bool;
      Ausencia_M375 : Bool;
      PresBloqueo_M375 : Bool;
      Galibo_M375 : Bool;
      PresPreparada_M375 : Bool;
      PresMultiple_M375 : Bool;
      Bit_07_M375 : Bool;
      RecepOK_M376 : Bool;
      PresNormal_M376 : Bool;
      Ausencia_M376 : Bool;
      PresBloqueo_M376 : Bool;
      Galibo_M376 : Bool;
      PresPreparada_M376 : Bool;
      PresMultiple_M376 : Bool;
      Bit_07_M376 : Bool;
      RecepOK_M377 : Bool;
      PresNormal_M377 : Bool;
      Ausencia_M377 : Bool;
      PresBloqueo_M377 : Bool;
      Galibo_M377 : Bool;
      PresPreparada_M377 : Bool;
      PresMultiple_M377 : Bool;
      Bit_07_M377 : Bool;
      RecepOK_M378 : Bool;
      PresNormal_M378 : Bool;
      Ausencia_M378 : Bool;
      PresBloqueo_M378 : Bool;
      Galibo_M378 : Bool;
      PresPreparada_M378 : Bool;
      PresMultiple_M378 : Bool;
      Bit_07_M378 : Bool;
      RecepOK_M379 : Bool;
      PresNormal_M379 : Bool;
      Ausencia_M379 : Bool;
      PresBloqueo_M379 : Bool;
      Galibo_M379 : Bool;
      PresPreparada_M379 : Bool;
      PresMultiple_M379 : Bool;
      Bit_07_M379 : Bool;
      RecepOK_M380 : Bool;
      PresNormal_M380 : Bool;
      Ausencia_M380 : Bool;
      PresBloqueo_M380 : Bool;
      Galibo_M380 : Bool;
      PresPreparada_M380 : Bool;
      PresMultiple_M380 : Bool;
      Bit_07_M380 : Bool;
      RecepOK_M381 : Bool;
      PresNormal_M381 : Bool;
      Ausencia_M381 : Bool;
      PresBloqueo_M381 : Bool;
      Galibo_M381 : Bool;
      PresPreparada_M381 : Bool;
      PresMultiple_M381 : Bool;
      Bit_07_M381 : Bool;
      RecepOK_M382 : Bool;
      PresNormal_M382 : Bool;
      Ausencia_M382 : Bool;
      PresBloqueo_M382 : Bool;
      Galibo_M382 : Bool;
      PresPreparada_M382 : Bool;
      PresMultiple_M382 : Bool;
      Bit_07_M382 : Bool;
      RecepOK_M383 : Bool;
      PresNormal_M383 : Bool;
      Ausencia_M383 : Bool;
      PresBloqueo_M383 : Bool;
      Galibo_M383 : Bool;
      PresPreparada_M383 : Bool;
      PresMultiple_M383 : Bool;
      Bit_07_M383 : Bool;
      RecepOK_M384 : Bool;
      PresNormal_M384 : Bool;
      Ausencia_M384 : Bool;
      PresBloqueo_M384 : Bool;
      Galibo_M384 : Bool;
      PresPreparada_M384 : Bool;
      PresMultiple_M384 : Bool;
      Bit_07_M384 : Bool;
      RecepOK_M385 : Bool;
      PresNormal_M385 : Bool;
      Ausencia_M385 : Bool;
      PresBloqueo_M385 : Bool;
      Galibo_M385 : Bool;
      PresPreparada_M385 : Bool;
      PresMultiple_M385 : Bool;
      Bit_07_M385 : Bool;
      RecepOK_M386 : Bool;
      PresNormal_M386 : Bool;
      Ausencia_M386 : Bool;
      PresBloqueo_M386 : Bool;
      Galibo_M386 : Bool;
      PresPreparada_M386 : Bool;
      PresMultiple_M386 : Bool;
      Bit_07_M386 : Bool;
      RecepOK_M387 : Bool;
      PresNormal_M387 : Bool;
      Ausencia_M387 : Bool;
      PresBloqueo_M387 : Bool;
      Galibo_M387 : Bool;
      PresPreparada_M387 : Bool;
      PresMultiple_M387 : Bool;
      Bit_07_M387 : Bool;
      RecepOK_M388 : Bool;
      PresNormal_M388 : Bool;
      Ausencia_M388 : Bool;
      PresBloqueo_M388 : Bool;
      Galibo_M388 : Bool;
      PresPreparada_M388 : Bool;
      PresMultiple_M388 : Bool;
      Bit_07_M388 : Bool;
      RecepOK_M389 : Bool;
      PresNormal_M389 : Bool;
      Ausencia_M389 : Bool;
      PresBloqueo_M389 : Bool;
      Galibo_M389 : Bool;
      PresPreparada_M389 : Bool;
      PresMultiple_M389 : Bool;
      Bit_07_M389 : Bool;
      RecepOK_M390 : Bool;
      PresNormal_M390 : Bool;
      Ausencia_M390 : Bool;
      PresBloqueo_M390 : Bool;
      Galibo_M390 : Bool;
      PresPreparada_M390 : Bool;
      PresMultiple_M390 : Bool;
      Bit_07_M390 : Bool;
      RecepOK_M391 : Bool;
      PresNormal_M391 : Bool;
      Ausencia_M391 : Bool;
      PresBloqueo_M391 : Bool;
      Galibo_M391 : Bool;
      PresPreparada_M391 : Bool;
      PresMultiple_M391 : Bool;
      Bit_07_M391 : Bool;
      RecepOK_M392 : Bool;
      PresNormal_M392 : Bool;
      Ausencia_M392 : Bool;
      PresBloqueo_M392 : Bool;
      Galibo_M392 : Bool;
      PresPreparada_M392 : Bool;
      PresMultiple_M392 : Bool;
      Bit_07_M392 : Bool;
      RecepOK_M393 : Bool;
      PresNormal_M393 : Bool;
      Ausencia_M393 : Bool;
      PresBloqueo_M393 : Bool;
      Galibo_M393 : Bool;
      PresPreparada_M393 : Bool;
      PresMultiple_M393 : Bool;
      Bit_07_M393 : Bool;
      RecepOK_M394 : Bool;
      PresNormal_M394 : Bool;
      Ausencia_M394 : Bool;
      PresBloqueo_M394 : Bool;
      Galibo_M394 : Bool;
      PresPreparada_M394 : Bool;
      PresMultiple_M394 : Bool;
      Bit_07_M394 : Bool;
      RecepOK_M395 : Bool;
      PresNormal_M395 : Bool;
      Ausencia_M395 : Bool;
      PresBloqueo_M395 : Bool;
      Galibo_M395 : Bool;
      PresPreparada_M395 : Bool;
      PresMultiple_M395 : Bool;
      Bit_07_M395 : Bool;
      RecepOK_M396 : Bool;
      PresNormal_M396 : Bool;
      Ausencia_M396 : Bool;
      PresBloqueo_M396 : Bool;
      Galibo_M396 : Bool;
      PresPreparada_M396 : Bool;
      PresMultiple_M396 : Bool;
      Bit_07_M396 : Bool;
      RecepOK_M397 : Bool;
      PresNormal_M397 : Bool;
      Ausencia_M397 : Bool;
      PresBloqueo_M397 : Bool;
      Galibo_M397 : Bool;
      PresPreparada_M397 : Bool;
      PresMultiple_M397 : Bool;
      Bit_07_M397 : Bool;
      RecepOK_M398 : Bool;
      PresNormal_M398 : Bool;
      Ausencia_M398 : Bool;
      PresBloqueo_M398 : Bool;
      Galibo_M398 : Bool;
      PresPreparada_M398 : Bool;
      PresMultiple_M398 : Bool;
      Bit_07_M398 : Bool;
      RecepOK_M399 : Bool;
      PresNormal_M399 : Bool;
      Ausencia_M399 : Bool;
      PresBloqueo_M399 : Bool;
      Galibo_M399 : Bool;
      PresPreparada_M399 : Bool;
      PresMultiple_M399 : Bool;
      Bit_07_M399 : Bool;
      RecepOK_M400 : Bool;
      PresNormal_M400 : Bool;
      Ausencia_M400 : Bool;
      PresBloqueo_M400 : Bool;
      Galibo_M400 : Bool;
      PresPreparada_M400 : Bool;
      PresMultiple_M400 : Bool;
      Bit_07_M400 : Bool;
      RecepOK_M401 : Bool;
      PresNormal_M401 : Bool;
      Ausencia_M401 : Bool;
      PresBloqueo_M401 : Bool;
      Galibo_M401 : Bool;
      PresPreparada_M401 : Bool;
      PresMultiple_M401 : Bool;
      Bit_07_M401 : Bool;
      RecepOK_M402 : Bool;
      PresNormal_M402 : Bool;
      Ausencia_M402 : Bool;
      PresBloqueo_M402 : Bool;
      Galibo_M402 : Bool;
      PresPreparada_M402 : Bool;
      PresMultiple_M402 : Bool;
      Bit_07_M402 : Bool;
      RecepOK_M403 : Bool;
      PresNormal_M403 : Bool;
      Ausencia_M403 : Bool;
      PresBloqueo_M403 : Bool;
      Galibo_M403 : Bool;
      PresPreparada_M403 : Bool;
      PresMultiple_M403 : Bool;
      Bit_07_M403 : Bool;
      RecepOK_M404 : Bool;
      PresNormal_M404 : Bool;
      Ausencia_M404 : Bool;
      PresBloqueo_M404 : Bool;
      Galibo_M404 : Bool;
      PresPreparada_M404 : Bool;
      PresMultiple_M404 : Bool;
      Bit_07_M404 : Bool;
      RecepOK_M405 : Bool;
      PresNormal_M405 : Bool;
      Ausencia_M405 : Bool;
      PresBloqueo_M405 : Bool;
      Galibo_M405 : Bool;
      PresPreparada_M405 : Bool;
      PresMultiple_M405 : Bool;
      Bit_07_M405 : Bool;
      RecepOK_M406 : Bool;
      PresNormal_M406 : Bool;
      Ausencia_M406 : Bool;
      PresBloqueo_M406 : Bool;
      Galibo_M406 : Bool;
      PresPreparada_M406 : Bool;
      PresMultiple_M406 : Bool;
      Bit_07_M406 : Bool;
      RecepOK_M407 : Bool;
      PresNormal_M407 : Bool;
      Ausencia_M407 : Bool;
      PresBloqueo_M407 : Bool;
      Galibo_M407 : Bool;
      PresPreparada_M407 : Bool;
      PresMultiple_M407 : Bool;
      Bit_07_M407 : Bool;
      RecepOK_M408 : Bool;
      PresNormal_M408 : Bool;
      Ausencia_M408 : Bool;
      PresBloqueo_M408 : Bool;
      Galibo_M408 : Bool;
      PresPreparada_M408 : Bool;
      PresMultiple_M408 : Bool;
      Bit_07_M408 : Bool;
      RecepOK_M409 : Bool;
      PresNormal_M409 : Bool;
      Ausencia_M409 : Bool;
      PresBloqueo_M409 : Bool;
      Galibo_M409 : Bool;
      PresPreparada_M409 : Bool;
      PresMultiple_M409 : Bool;
      Bit_07_M409 : Bool;
      RecepOK_M410 : Bool;
      PresNormal_M410 : Bool;
      Ausencia_M410 : Bool;
      PresBloqueo_M410 : Bool;
      Galibo_M410 : Bool;
      PresPreparada_M410 : Bool;
      PresMultiple_M410 : Bool;
      Bit_07_M410 : Bool;
      RecepOK_M411 : Bool;
      PresNormal_M411 : Bool;
      Ausencia_M411 : Bool;
      PresBloqueo_M411 : Bool;
      Galibo_M411 : Bool;
      PresPreparada_M411 : Bool;
      PresMultiple_M411 : Bool;
      Bit_07_M411 : Bool;
      RecepOK_M412 : Bool;
      PresNormal_M412 : Bool;
      Ausencia_M412 : Bool;
      PresBloqueo_M412 : Bool;
      Galibo_M412 : Bool;
      PresPreparada_M412 : Bool;
      PresMultiple_M412 : Bool;
      Bit_07_M412 : Bool;
      RecepOK_M413 : Bool;
      PresNormal_M413 : Bool;
      Ausencia_M413 : Bool;
      PresBloqueo_M413 : Bool;
      Galibo_M413 : Bool;
      PresPreparada_M413 : Bool;
      PresMultiple_M413 : Bool;
      Bit_07_M413 : Bool;
      RecepOK_M414 : Bool;
      PresNormal_M414 : Bool;
      Ausencia_M414 : Bool;
      PresBloqueo_M414 : Bool;
      Galibo_M414 : Bool;
      PresPreparada_M414 : Bool;
      PresMultiple_M414 : Bool;
      Bit_07_M414 : Bool;
      RecepOK_M415 : Bool;
      PresNormal_M415 : Bool;
      Ausencia_M415 : Bool;
      PresBloqueo_M415 : Bool;
      Galibo_M415 : Bool;
      PresPreparada_M415 : Bool;
      PresMultiple_M415 : Bool;
      Bit_07_M415 : Bool;
      RecepOK_M416 : Bool;
      PresNormal_M416 : Bool;
      Ausencia_M416 : Bool;
      PresBloqueo_M416 : Bool;
      Galibo_M416 : Bool;
      PresPreparada_M416 : Bool;
      PresMultiple_M416 : Bool;
      Bit_07_M416 : Bool;
      RecepOK_M417 : Bool;
      PresNormal_M417 : Bool;
      Ausencia_M417 : Bool;
      PresBloqueo_M417 : Bool;
      Galibo_M417 : Bool;
      PresPreparada_M417 : Bool;
      PresMultiple_M417 : Bool;
      Bit_07_M417 : Bool;
      RecepOK_M418 : Bool;
      PresNormal_M418 : Bool;
      Ausencia_M418 : Bool;
      PresBloqueo_M418 : Bool;
      Galibo_M418 : Bool;
      PresPreparada_M418 : Bool;
      PresMultiple_M418 : Bool;
      Bit_07_M418 : Bool;
      RecepOK_M419 : Bool;
      PresNormal_M419 : Bool;
      Ausencia_M419 : Bool;
      PresBloqueo_M419 : Bool;
      Galibo_M419 : Bool;
      PresPreparada_M419 : Bool;
      PresMultiple_M419 : Bool;
      Bit_07_M419 : Bool;
      RecepOK_M420 : Bool;
      PresNormal_M420 : Bool;
      Ausencia_M420 : Bool;
      PresBloqueo_M420 : Bool;
      Galibo_M420 : Bool;
      PresPreparada_M420 : Bool;
      PresMultiple_M420 : Bool;
      Bit_07_M420 : Bool;
      RecepOK_M421 : Bool;
      PresNormal_M421 : Bool;
      Ausencia_M421 : Bool;
      PresBloqueo_M421 : Bool;
      Galibo_M421 : Bool;
      PresPreparada_M421 : Bool;
      PresMultiple_M421 : Bool;
      Bit_07_M421 : Bool;
      RecepOK_M422 : Bool;
      PresNormal_M422 : Bool;
      Ausencia_M422 : Bool;
      PresBloqueo_M422 : Bool;
      Galibo_M422 : Bool;
      PresPreparada_M422 : Bool;
      PresMultiple_M422 : Bool;
      Bit_07_M422 : Bool;
      RecepOK_M423 : Bool;
      PresNormal_M423 : Bool;
      Ausencia_M423 : Bool;
      PresBloqueo_M423 : Bool;
      Galibo_M423 : Bool;
      PresPreparada_M423 : Bool;
      PresMultiple_M423 : Bool;
      Bit_07_M423 : Bool;
      RecepOK_M424 : Bool;
      PresNormal_M424 : Bool;
      Ausencia_M424 : Bool;
      PresBloqueo_M424 : Bool;
      Galibo_M424 : Bool;
      PresPreparada_M424 : Bool;
      PresMultiple_M424 : Bool;
      Bit_07_M424 : Bool;
      RecepOK_M425 : Bool;
      PresNormal_M425 : Bool;
      Ausencia_M425 : Bool;
      PresBloqueo_M425 : Bool;
      Galibo_M425 : Bool;
      PresPreparada_M425 : Bool;
      PresMultiple_M425 : Bool;
      Bit_07_M425 : Bool;
      RecepOK_M426 : Bool;
      PresNormal_M426 : Bool;
      Ausencia_M426 : Bool;
      PresBloqueo_M426 : Bool;
      Galibo_M426 : Bool;
      PresPreparada_M426 : Bool;
      PresMultiple_M426 : Bool;
      Bit_07_M426 : Bool;
      RecepOK_M427 : Bool;
      PresNormal_M427 : Bool;
      Ausencia_M427 : Bool;
      PresBloqueo_M427 : Bool;
      Galibo_M427 : Bool;
      PresPreparada_M427 : Bool;
      PresMultiple_M427 : Bool;
      Bit_07_M427 : Bool;
      RecepOK_M428 : Bool;
      PresNormal_M428 : Bool;
      Ausencia_M428 : Bool;
      PresBloqueo_M428 : Bool;
      Galibo_M428 : Bool;
      PresPreparada_M428 : Bool;
      PresMultiple_M428 : Bool;
      Bit_07_M428 : Bool;
      RecepOK_M429 : Bool;
      PresNormal_M429 : Bool;
      Ausencia_M429 : Bool;
      PresBloqueo_M429 : Bool;
      Galibo_M429 : Bool;
      PresPreparada_M429 : Bool;
      PresMultiple_M429 : Bool;
      Bit_07_M429 : Bool;
      RecepOK_M430 : Bool;
      PresNormal_M430 : Bool;
      Ausencia_M430 : Bool;
      PresBloqueo_M430 : Bool;
      Galibo_M430 : Bool;
